# B&R Automation Studio project A2019059_Linka_Power_CP (part 26)

#### Main.st - Init, cyclic, exit code
```iecst
PROGRAM _INIT
	TprazdnyZasobnik.PT:=T#2000ms;
	TakumulaciaPlna.PT:=T#1000ms;
	TvytvorenieVakua.PT:=T#200ms;
	TodvetranieVakua.PT:=T#200ms;
	ToneskorenieVysunutia.PT:= T#500ms;
	ToneskorenieZasunutia.PT:= T#500ms;
	TvyfukovaniePredVibrovanim.PT:= T#1000ms;
    Tvibrovanie.PT:=T#3000ms;
    Stav_MaticaPripravena:= FALSE;
    TpodaniaSkrutky.PT:= T#1000ms;
    TpredMaticaPripravena.PT:= T#1000ms;
    TpripravaMatice.PT:= T#2000ms;
    TvypnutieOfuku.PT:= T#2000ms;
END_PROGRAM

PROGRAM _CYCLIC
	(********************Mapovanie IN/OUT********************************)

	SkrutkovaciSet.Manual:= P2_SkrutkovacMatic.SkrutkovaciSet_MaticaM4.Manual;
	SkrutkovaciSet.Automat:= P2_SkrutkovacMatic.SkrutkovaciSet_MaticaM4.Automat;
	SkrutkovaciSet.SkrutkaOdobrata:= P2_SkrutkovacMatic.SkrutkovaciSet_MaticaM4.MaticaM4_Odobrata;
	P2_SkrutkovacMatic.SkrutkovaciSet_MaticaM4.MaticaM4_Pripravena:= SkrutkovaciSet.SkrutkaPripravena;

	SkrutkovaciSet.Vreteno.IN.DeptControl;
	SkrutkovaciSet.Vreteno.IN.PushClinderAR:= P2_SkrutkovacMatic.IN.DavkMatic_VYSUNUTY_IS26;
	SkrutkovaciSet.Vreteno.IN.PushClinderGR:= P2_SkrutkovacMatic.IN.DavkMatic_ZASUNUTY_IS25;
	SkrutkovaciSet.Vreteno.IN.ReturnStroke:= P2_SkrutkovacMatic.IN.SkrutkMatic_ZASUNUTY_MS9;
	SkrutkovaciSet.Vreteno.IN.ScrewControl:= P2_SkrutkovacMatic.IN.DavkMatic_PritomnostMatice_OS2;
	SkrutkovaciSet.Vreteno.IN.ScrewMeasurement:= P2_SkrutkovacMatic.IN.OddelMatic_MaticaPresla_IS24;
	SkrutkovaciSet.Vreteno.IN.ScrewMeasurementPushCylinder:= P2_SkrutkovacMatic.IN.DavkMatic_MaticaPresla_IS27;

	P2_SkrutkovacMatic.OUT.PosuvacMatic_PosunMaticu_YV68:=SkrutkovaciSet.Vreteno.OUT.PushCylinder;

	SkrutkovaciSet.Zasobnik.IN.AccumulationSwitch:= P2_SkrutkovacMatic.IN.ZasobMatic_ListaPLNA_OS1;
	SkrutkovaciSet.Zasobnik.IN.FeederLevelControl:= P2_SkrutkovacMatic.IN.ZasobMatic_PRAZDNY_IS23;
	SkrutkovaciSet.Zasobnik.IN.EscapementAR:= P2_SkrutkovacMatic.IN.OddelMatic_Otoceny_VPRED_MS59;
	SkrutkovaciSet.Zasobnik.IN.EscapementGR:= P2_SkrutkovacMatic.IN.OddelMatic_Otoceny_VZAD_MS58;

	P2_SkrutkovacMatic.OUT.ZasobMatic_Ofuk_RUN_YV63:=SkrutkovaciSet.Zasobnik.OUT.BlowOff;
	P2_SkrutkovacMatic.OUT.OddelMatic_PosunMaticu_YV69:=SkrutkovaciSet.Zasobnik.OUT.Escapement;
	P2_SkrutkovacMatic.OUT.OddelMatic_NastrelMaticu_YV65:=SkrutkovaciSet.Zasobnik.OUT.FeedAir;
	P2_SkrutkovacMatic.OUT.ZasobMatic_OfukTried_RUN_YV64:=SkrutkovaciSet.Zasobnik.OUT.SortingAir;
	P2_SkrutkovacMatic.OUT.ZasobMatic_Vibrovanie_RUN_FM1:=SkrutkovaciSet.Zasobnik.OUT.StartA20;

	IF P2_SkrutkovacMatic.SkrutkovaciSet_MaticaM4.Reset THEN
		SkrutkovaciSet.VretenoFaza:=0;
		P2_SkrutkovacMatic.SkrutkovaciSet_MaticaM4.Reset:= FALSE;
	END_IF

	(********************Časáky********************************)
	TprazdnyZasobnik();
	TakumulaciaPlna();
	TvytvorenieVakua();
	TodvetranieVakua();
	ToneskorenieVysunutia();
    ToneskorenieZasunutia();
    Tvibrovanie();
    TvyfukovaniePredVibrovanim();
    TpodaniaSkrutky();
    TpredMaticaPripravena();
    TpripravaMatice();
    TvypnutieOfuku();
	(********************Zásobnik********************************)

	//kontrola akumulacie
	IF SkrutkovaciSet.Zasobnik.IN.AccumulationSwitch=1 THEN
		TakumulaciaPlna.IN:=1;
	ELSE
		TakumulaciaPlna.IN:=0;
	END_IF

	//kontrola naplnenia zasobnika
	IF SkrutkovaciSet.Zasobnik.IN.FeederLevelControl=1 THEN
		TprazdnyZasobnik.IN:=1;
	ELSE
		TprazdnyZasobnik.IN:=0;
	END_IF

    IF ZapniHrniec THEN
        TvyfukovaniePredVibrovanim.IN:= 1;
    ELSE
		TvyfukovaniePredVibrovanim.IN:= 0;
	END_IF

	IF ZapniHrniec AND TvyfukovaniePredVibrovanim.Q THEN
        SkrutkovaciSet.Zasobnik.OUT.StartA20:=1;
        Tvibrovanie.IN:=1;
	ELSE
        SkrutkovaciSet.Zasobnik.OUT.StartA20:=0;
        Tvibrovanie.IN:=0;
	END_IF

    IF Tvibrovanie.Q=1 THEN
        IF TakumulaciaPlna.Q=1 AND NOT P2_SkrutkovacMatic.RR_ZapniHrniec THEN
            ZapniHrniec:= 0;
        END_IF
    END_IF

    //Zapnutie hrnca v ručnom režime//
    IF EDGEPOS(P2_SkrutkovacMatic.RR_ZapniHrniec) THEN
        ZapniHrniec:= TRUE;
    END_IF
    IF EDGENEG(P2_SkrutkovacMatic.RR_ZapniHrniec) THEN
        ZapniHrniec:= FALSE;
    END_IF

    //Ovládanie vzduchov zásobníka//
    IF ZapniHrniec THEN
        IF TakumulaciaPlna.Q=1 THEN
            SkrutkovaciSet.Zasobnik.OUT.BlowOff:=1;
        ELSE
            SkrutkovaciSet.Zasobnik.OUT.BlowOff:=0;
        END_IF
        SkrutkovaciSet.Zasobnik.OUT.SortingAir:= 1;
    ELSE
        SkrutkovaciSet.Zasobnik.OUT.BlowOff:=0;
    END_IF

    IF NOT SkrutkovaciSet.Zasobnik.OUT.StartA20 AND NOT ZapniHrniec THEN
        TvypnutieOfuku.IN:= 1;
    ELSE
        TvypnutieOfuku.IN:= 0;
    END_IF

    IF EDGEPOS(TvypnutieOfuku.Q) THEN
        SkrutkovaciSet.Zasobnik.OUT.SortingAir:= 0;
    END_IF

	(********************Vreteno********************************)
	CASE SkrutkovaciSet.VretenoFaza OF
		0: SkrutkovaciSet.VretenoStatus:="Vypnute";
			SkrutkovaciSet.Vreteno.OUT.CounterBlast:=0;
			SkrutkovaciSet.Vreteno.OUT.Spindle:=0;

			SkrutkovaciSet.Zasobnik.OUT.Escapement:=0;
			SkrutkovaciSet.Zasobnik.OUT.FeedAir:=0;

			SkrutkovaciSet.Zasobnik.OUT.StartA20:=0;

			SkrutkovaciSet.SkrutkaPripravena:=0;

			TprazdnyZasobnik.IN:=0;
			TakumulaciaPlna.IN:=0;
			TvytvorenieVakua.IN:=0;
			TodvetranieVakua.IN:=0;
			ToneskorenieVysunutia.IN:=0;
            ToneskorenieZasunutia.IN:= 0;
            TpodaniaSkrutky.IN:= 0;
            TpredMaticaPripravena.IN:= 0;
            TpripravaMatice.IN:= 0;
			ZapniHrniec:= 0;
			SkrutkovaciSet.VretenoFaza:=1;

		1: SkrutkovaciSet.VretenoStatus:="Inicializacia: cakam na povel";
			IF SkrutkovaciSet.Automat=1 THEN
				SkrutkovaciSet.SkrutkaPripravena:=0;
				SkrutkovaciSet.VretenoFaza:=2;
			ELSIF SkrutkovaciSet.Manual=1 THEN
				SkrutkovaciSet.VretenoFaza:=250;
			ELSIF P2_SkrutkovacMatic.RR_PodajMaticu THEN
				Stav_MaticaPripravena:= FALSE;
				SkrutkovaciSet.VretenoFaza:=2;
			END_IF

		2: SkrutkovaciSet.VretenoStatus:="Inicializacia: cakam na snimac koliska vo vstupnej polohe";
			SkrutkovaciSet.Zasobnik.OUT.Escapement:=0;
			IF SkrutkovaciSet.Zasobnik.IN.EscapementGR=1 THEN
				SkrutkovaciSet.Zasobnik.OUT.FeedAir:=1;
				SkrutkovaciSet.VretenoFaza:=3;
			END_IF

		3: SkrutkovaciSet.VretenoStatus:="Inicializacia: Cakam na snimac: podavaci piest zasunuty";
			SkrutkovaciSet.Vreteno.OUT.PushCylinder:=0;
			IF SkrutkovaciSet.Vreteno.IN.PushClinderGR=1 THEN
				SkrutkovaciSet.VretenoFaza:=4;
			END_IF

		4: SkrutkovaciSet.VretenoStatus:="Inicializacia: kontrolujem pritomnost matky";
			IF SkrutkovaciSet.Vreteno.IN.ScrewControl=1 THEN
				SkrutkovaciSet.Zasobnik.OUT.FeedAir:=0;
				SkrutkovaciSet.VretenoFaza:=100;
			ELSE
				SkrutkovaciSet.VretenoFaza:=5;
			END_IF

		5: SkrutkovaciSet.VretenoStatus:="Inicializacia: Cakam na snimac: podavaci piest vysunuty";
			SkrutkovaciSet.Vreteno.OUT.PushCylinder:=1;
			IF SkrutkovaciSet.Vreteno.IN.PushClinderAR=1 THEN
				SkrutkovaciSet.VretenoFaza:=6;
			END_IF

		6: SkrutkovaciSet.VretenoStatus:="Inicializacia: Cakam na snimac: podavaci piest zasunuty";
			SkrutkovaciSet.Vreteno.OUT.PushCylinder:=0;
			IF SkrutkovaciSet.Vreteno.IN.PushClinderGR=1 THEN
				SkrutkovaciSet.VretenoFaza:=7;
			END_IF

		7: SkrutkovaciSet.VretenoStatus:="Inicializacia: kontrolujem pritomnost matky";
			IF SkrutkovaciSet.Vreteno.IN.ScrewControl=1 THEN
				SkrutkovaciSet.Vreteno.OUT.Vacuum:=1;
				SkrutkovaciSet.Zasobnik.OUT.FeedAir:=0;
				SkrutkovaciSet.VretenoFaza:=100;
			ELSE
				SkrutkovaciSet.Zasobnik.OUT.FeedAir:=0;
				SkrutkovaciSet.VretenoFaza:=150;
			END_IF

		100: SkrutkovaciSet.VretenoStatus:="Pripravene: cakam na povel";
			SkrutkovaciSet.SkrutkaPripravena:=1;
			IF P2_SkrutkovacMatic.RR_PodajMaticu THEN
				SkrutkovaciSet.Vreteno.OUT.Vacuum:=0;
				SkrutkovaciSet.SkrutkaPripravena:=0;
				P2_SkrutkovacMatic.RR_PodajMaticu:= FALSE;
                SkrutkovaciSet.VretenoFaza:=0;
			END_IF

			IF SkrutkovaciSet.SkrutkaOdobrata=1 THEN
				SkrutkovaciSet.Vreteno.OUT.Vacuum:=0;
				SkrutkovaciSet.SkrutkaPripravena:=0;
				SkrutkovaciSet.VretenoFaza:=101;
			END_IF

		101: SkrutkovaciSet.VretenoStatus:="Cakam kym zmizne signal skrutka odobrata";
			SkrutkovaciSet.SkrutkaPripravena:=0;
			IF SkrutkovaciSet.SkrutkaOdobrata=0 THEN
				SkrutkovaciSet.VretenoFaza:=150;
			END_IF

		150: SkrutkovaciSet.VretenoStatus:="Cakam kym zasobnik pripravy skrutku";
			ZapniHrniec:= 1;
            IF TakumulaciaPlna.Q=1 AND SkrutkovaciSet.Zasobnik.OUT.StartA20 THEN
                TpodaniaSkrutky.IN:= 1;
            END_IF

            IF TpodaniaSkrutky.Q THEN
                TpodaniaSkrutky.IN:= 0;
                SkrutkovaciSet.VretenoFaza:=151;
			END_IF

		151: SkrutkovaciSet.VretenoStatus:="Cakam na snimac: koliska vo vystupnej polohe";
			SkrutkovaciSet.Zasobnik.OUT.Escapement:=1;
			IF SkrutkovaciSet.Zasobnik.IN.EscapementAR=1 THEN
				SkrutkovaciSet.VretenoFaza:=152;
			END_IF

		152: SkrutkovaciSet.VretenoStatus:="Cakam na snimac: skrutka presla hadicou za zasobnikom";

            TpripravaMatice.IN:=1;
			IF SkrutkovaciSet.Vreteno.IN.ScrewMeasurement=1 THEN
                SkrutkovaciSet.Zasobnik.OUT.FeedAir:=1;
                TpripravaMatice.IN:=0;
                SkrutkovaciSet.VretenoFaza:=153;
            ELSIF TpripravaMatice.Q THEN
                TpripravaMatice.IN:=0;
                SkrutkovaciSet.Zasobnik.OUT.Escapement:=0;
                SkrutkovaciSet.VretenoFaza:=150;
			END_IF

		153: SkrutkovaciSet.VretenoStatus:="Cakam na snimac: skrutka presla hadicou pred piestom";
			SkrutkovaciSet.Zasobnik.OUT.FeedAir:=1;
			IF SkrutkovaciSet.Vreteno.IN.ScrewMeasurementPushCylinder=1 THEN
				ToneskorenieVysunutia.IN:= 1;
			END_IF
			IF ToneskorenieVysunutia.Q THEN
				ToneskorenieVysunutia.IN:= 0;
				SkrutkovaciSet.Zasobnik.OUT.FeedAir:=0;
				SkrutkovaciSet.VretenoFaza:=154;
			END_IF

		154: SkrutkovaciSet.VretenoStatus:="Cakam na snimac: podavaci piest vysunuty";
			SkrutkovaciSet.Vreteno.OUT.PushCylinder:=1;
			SkrutkovaciSet.Vreteno.OUT.Vacuum:=1;
			IF SkrutkovaciSet.Vreteno.IN.PushClinderAR=1 THEN
				SkrutkovaciSet.Zasobnik.OUT.FeedAir:=0;
				SkrutkovaciSet.VretenoFaza:=155;
			END_IF

		155: SkrutkovaciSet.VretenoStatus:="Cakam na snimac: matka v hlavici";
			ToneskorenieZasunutia.IN:= SkrutkovaciSet.Vreteno.IN.ScrewControl;
			IF SkrutkovaciSet.Vreteno.IN.ScrewControl=1 AND ToneskorenieZasunutia.Q THEN
				ToneskorenieZasunutia.IN:= 0;
				SkrutkovaciSet.VretenoFaza:=156;
			END_IF

		156: SkrutkovaciSet.VretenoStatus:="Cakam na snimac: podavaci piest zasunuty";
			SkrutkovaciSet.Vreteno.OUT.PushCylinder:=0;
			IF SkrutkovaciSet.Vreteno.IN.PushClinderGR=1 THEN
				SkrutkovaciSet.VretenoFaza:=157;
			END_IF

		157: SkrutkovaciSet.VretenoStatus:="Cakam na snimac: koliska vo vstupnej polohe";
			SkrutkovaciSet.Zasobnik.OUT.Escapement:=0;
			IF SkrutkovaciSet.Zasobnik.IN.EscapementGR=1 THEN
				SkrutkovaciSet.VretenoFaza:=158;
			END_IF

		158: SkrutkovaciSet.VretenoStatus:="Novy cyklus";
			SkrutkovaciSet.VretenoFaza:=100;
	END_CASE

END_PROGRAM

PROGRAM _EXIT
	(* Insert code here *)

END_PROGRAM
```

#### Types.typ - Local data types
```iecst
TYPE
	SkrutkovaciSetStruc : 	STRUCT
		VretenoStatus : WSTRING[80];
		VretenoFaza : USINT;
		Zasobnik : ZasobnikStruc;
		Vreteno : VretenoStruc;
		SkrutkaOdobrata : BOOL;
		SkrutkaPripravena : BOOL;
		Manual : BOOL;
		PodajSrobu : BOOL;
		CistenieVykonane : BOOL;
		VykonajCistenie : BOOL;
		Automat : BOOL;
	END_STRUCT;
	INzasobnik : 	STRUCT
		EscapementGR : BOOL;
		EscapementAR : BOOL;
		AccumulationSwitch : BOOL; (*Snimac zaplnenia S25*)
		FeederLevelControl : BOOL; (*Hladina v zasobniku S20*)
	END_STRUCT;
	OUTzasobnik : 	STRUCT
		StartA20 : BOOL; (*Zapnutie vibrovania A20*)
		Escapement : BOOL; (*Pustanie matky do hadice Y22*)
		FeedAir : BOOL; (*Strielanie do hadice Y21*)
		SortingAir : BOOL; (*Triedenie kusov Y30*)
		BlowOff : BOOL; (*Zhadzovanie kusov Y25*)
	END_STRUCT;
	INvreteno : 	STRUCT
		ReturnStroke : BOOL; (*Vreteno zasunute S01*)
		DeptControl : BOOL; (*Vreteno vysunute S02*)
		PushClinderGR : BOOL; (*Posuvaci valec v domovskej  polohe S11*)
		PushClinderAR : BOOL; (*Posuvaci valec v pracovnej polohe S10*)
		ScrewMeasurement : BOOL; (*Kontrola matice v hadici S21*)
		ScrewMeasurementPushCylinder : BOOL; (*Kontrola matice v posuvacom valci S06*)
		ScrewControl : BOOL; (*Kontrola matice vo vretene S14*)
	END_STRUCT;
	OUTvreteno : 	STRUCT
		Spindle : BOOL; (*Vysunutie vretena Y02*)
		Vacuum : BOOL; (*Pridrzanie skrutky Y15*)
		PushCylinder : BOOL; (*Posunutie z hadice do hlavy Y10*)
		CounterBlast : BOOL; (*Uvolnenie skrutky Y16*)
	END_STRUCT;
	VretenoStruc : 	STRUCT
		OUT : OUTvreteno;
		IN : INvreteno;
	END_STRUCT;
	ZasobnikStruc : 	STRUCT
		OUT : OUTzasobnik;
		IN : INzasobnik;
	END_STRUCT;
END_TYPE
```

#### Variables.var - Local variables
```iecst
VAR
	TvytvorenieVakua : TON;
	TodvetranieVakua : TON;
	TprazdnyZasobnik : TON;
	TakumulaciaPlna : TON;
	ToneskorenieVysunutia : TON;
	ToneskorenieZasunutia : TON;
	SkrutkovaciSet : SkrutkovaciSetStruc;
	Stav_MaticaPripravena : BOOL;
	TvyfukovaniePredVibrovanim : TON;
	ZapniHrniec : BOOL;
	TpodaniaSkrutky : TON;
	Tvibrovanie : TON;
	TpredMaticaPripravena : TON;
	TpripravaMatice : TON;
	TvypnutieOfuku : TON;
END_VAR
```

### Program Logical/Program/Pracovisko_2/P2_StoperSrobovania (IEC)

#### Main.st - Init, cyclic, exit code
```iecst
PROGRAM _INIT
    Triger_0:= FALSE;
    Triger_1:= FALSE;

END_PROGRAM

PROGRAM _CYCLIC

	//Volanie funkcie SequenceControl//
    SequenceControl(SC:= SC_P2_StoperSrobovania);

    //Volanie podprogramov//
    OvlCentrovacky;
    IOLinkKomunikacia;

    //Reset sekcie //
    IF P2_StoperSrobovania.Reset THEN
        SC_P2_StoperSrobovania.Step:= 0;
        P2_StoperSrobovania.Reset:= FALSE;
    END_IF

    IF NOT Safety.STAV.P2_ZonaBunky_AKTIVNA AND NOT P2_StoperSrobovania.Automat THEN
        SC_P2_StoperSrobovania.Step:= 0;
    END_IF

    IF NOT Safety.STAV.P2_ZonaBunky_AKTIVNA AND NOT Triger_0 THEN
        Triger_0:= TRUE;
        IF P2_StoperSrobovania.IN.PritomnostPaletky_S8 AND P2_StoperSrobovania.Automat THEN
            IF NOT Paletka[i].VnutornyStav.KomunikaciaOtvorena THEN
                SC_P2_StoperSrobovania.ResetStep:= TRUE;
                SC_P2_StoperSrobovania.Step:= 0;
            ELSIF Paletka[i].VnutornyStav.KomunikaciaUzavreta THEN
                SC_P2_StoperSrobovania.ResetStep:= TRUE;
                SC_P2_StoperSrobovania.Step:= 0;
            ELSIF Paletka[i].VnutornyStav.CinnostSpustena THEN
                Paletka[i].PAR.StavPowerCP:= 'FAIL';
                Paletka[i].PAR.StavPaletky:= 'NG';
                P2_StoperSrobovania.KoniecCyklu:= TRUE;
                SC_P2_StoperSrobovania.ResetStep:= TRUE;
                SC_P2_StoperSrobovania.Step:= 550;
            ELSIF Paletka[i].VnutornyStav.KomunikaciaOtvorena THEN
                Paletka[i].PAR.StavPowerCP:= 'FAIL';
                Paletka[i].PAR.StavPaletky:= 'NG';
                P2_StoperSrobovania.KoniecCyklu:= TRUE;
                SC_P2_StoperSrobovania.ResetStep:= TRUE;
                SC_P2_StoperSrobovania.Step:= 550;
            END_IF
        END_IF
    END_IF

    IF Safety.STAV.P2_ZonaBunky_AKTIVNA THEN
        Triger_0:= FALSE;
    END_IF

    //Porucha stanice//
    IF P2_PoruchaST3 AND NOT Triger_1 THEN
        Triger_1:= TRUE;
        IF P2_StoperSrobovania.IN.PritomnostPaletky_S8 AND P2_StoperSrobovania.Automat THEN
            SC_P2_Srobovanie.Step:= 0;
            IF NOT Paletka[i].VnutornyStav.KomunikaciaOtvorena THEN
                SC_P2_StoperSrobovania.ResetStep:= TRUE;
                SC_P2_StoperSrobovania.Step:= 0;
            ELSIF Paletka[i].VnutornyStav.KomunikaciaUzavreta THEN
                SC_P2_StoperSrobovania.ResetStep:= TRUE;
                SC_P2_StoperSrobovania.Step:= 0;
            ELSIF Paletka[i].VnutornyStav.CinnostSpustena THEN
                Paletka[i].PAR.StavPowerCP:= 'FAIL';
                Paletka[i].PAR.StavPaletky:= 'NG';
                P2_StoperSrobovania.KoniecCyklu:= TRUE;
                SC_P2_StoperSrobovania.ResetStep:= TRUE;
                SC_P2_StoperSrobovania.Step:= 550;
            ELSIF Paletka[i].VnutornyStav.KomunikaciaOtvorena THEN
                Paletka[i].PAR.StavPowerCP:= 'FAIL';
                Paletka[i].PAR.StavPaletky:= 'NG';
                P2_StoperSrobovania.KoniecCyklu:= TRUE;
                SC_P2_StoperSrobovania.ResetStep:= TRUE;
                SC_P2_StoperSrobovania.Step:= 550;
            END_IF
        ELSE
            SC_P2_StoperSrobovania.ResetStep:= TRUE;
            SC_P2_StoperSrobovania.Step:= 0;
        END_IF
    END_IF

    IF NOT P2_PoruchaST3 THEN
        Triger_1:= FALSE;
    END_IF

    CASE SC_P2_StoperSrobovania.Step OF

        0:
            SC_P2_StoperSrobovania.StepName:='0 - Nulovanie';
            SC_OvlCentrovacky.Step:= 0;
            P2_StoperSrobovania.Automat:= FALSE;
            P2_StoperSrobovania.KoniecCyklu:= FALSE;
            P2_StoperSrobovania.Manual:= FALSE;
            P2_StoperSrobovania.STAV.PoINIT:= FALSE;
            P2_StoperSrobovania.OUT.ZasunStoper_YV56:= FALSE;
            P2_StoperSrobovania.OUT.KOM_4F_ZasrobujLavuSkrutkuM4:= FALSE;
            P2_StoperSrobovania.OUT.KOM_4F_ZasrobujPravuSkrutkuM4:= FALSE;
            P2_StoperSrobovania.OUT.KOM_4F_ZasrobujLavuSkrutkuM6:= FALSE;
            P2_StoperSrobovania.OUT.KOM_4F_ZasrobujPravuSkrutkuM6:= FALSE;
            P2_StoperSrobovania.OUT.KOM_5F_ZasrobujLavuSkrutkuM4:= FALSE;
            P2_StoperSrobovania.OUT.KOM_5F_ZasrobujPravuSkrutkuM4:= FALSE;
            P2_StoperSrobovania.OUT.KOM_5F_ZasrobujLavuSkrutkuM6:= FALSE;
            P2_StoperSrobovania.OUT.KOM_5F_ZasrobujPravuSkrutkuM6:= FALSE;
            P2_StoperSrobovania.OUT.KOM_5H_ZasrobujLavuSkrutkuM5:= FALSE;
            P2_StoperSrobovania.OUT.KOM_5H_ZasrobujPravuSkrutkuM5:= FALSE;
            P2_StoperSrobovania.OUT.KOM_5H_ZasrobujSkrutkuM4:= FALSE;
            P2_StoperSrobovania.OUT.KOM_PresunManipulator_DOPREDU:= FALSE;
            P2_StoperSrobovania.OUT.KOM_PresunManipulator_DOZADU:= FALSE;
            P2_Srobovanie.OUT.KOM_Srobovanie_Ukoncene:= FALSE;
            P2_Srobovanie.OUT.KOM_PresunVPRED_Ukonceny:= FALSE;
            P2_Srobovanie.OUT.KOM_PresunVZAD_Ukonceny:= FALSE;
            P2_Robot.KOM_OUT.Odober_Busbary4F:= FALSE;
            P2_Robot.KOM_OUT.Odober_Busbary5F:= FALSE;
            P2_Robot.KOM_OUT.Odober_Busbary5H:= FALSE;
            P2_Robot.KOM_OUT.Poloz_Busbary4F:= FALSE;
            P2_Robot.KOM_OUT.Poloz_Busbary5F:= FALSE;
            P2_Robot.KOM_OUT.Poloz_Busbary5H:= FALSE;
            P2_Robot.KOM_OUT.Dotlac_Filter5H:= FALSE;
            P2_Robot.KOM_OUT.Odparkovanie:= FALSE;
            P2_Robot.KOM_OUT.Presun_CakaciaPozicia:= FALSE;
            P2_Robot.KOM_OUT.UvolniBusbary:= FALSE;
            P2_Robot.KOM_OUT.Dotlac_Filter5H:= FALSE;
            P2_Robot.KOM_OUT.ZmenaGripra_Cistenie:= FALSE;
            CAM10.CMD.Triger:= FALSE;
            CAM10.STAV.Results_READY:= FALSE;
            FTP_CAM10.CMD.OdosliFotku:= FALSE;
            FTP_CAM10.CMD.VymazFotku:= FALSE;
            P2_StoperSrobovania.STAV.KOM_PLC_OdoslanieFotiek_OK:= FALSE;
            P2_StoperSrobovania.STAV.KOM_PLC_VymazanieFotiek_OK:= FALSE;
            TRCB_P2_Srobovanie_ST5.CMD.VyziadajStavPaletky_TYP1:= FALSE;
            TRCB_P2_Srobovanie_ST5.CMD.PriradQRkodFiltra_TYP3:= FALSE;
            TRCB_P2_Srobovanie_ST5.CMD.OdosliStavPaletky_TYP2:= FALSE;
            PrecitaneCisloPaletky:= '';
            P2_Srobov_ManipulaciaUkoncena:= FALSE;
            PocetDopytovNaServer:= 0;
            Taktime_Srobovanie_ST5.CMD.START_Merania_1:= FALSE;
            Taktime_Srobovanie_ST5.CMD.START_Merania_2:= FALSE;
            P2_StoperSrobovania.STAV.PrebiehaVyvezeniePaletky:= FALSE;
            P2_Srobov_KAM_Result_Ignoruj:= FALSE;
            P2_Srobov_CakaNaKameru:= FALSE;
            P2_StoperSrobovania.STAV.Porucha:= FALSE;
            TestovaciKus:= FALSE;
            Revork:= FALSE;
            P2_Robot.STAV.Srobovanie_PrebiehaManipulacia:= FALSE;
            CisloFotky:= 0;
            P2_Srobov_KAM_Result_OK:= FALSE;
            P2_Srobov_KAM_Result_NG:= FALSE;
            P2_Vizu.ZobrazHL1_ST5:= FALSE;
            P2_Vizu.ZobrazHL2_ST5:= FALSE;
            P2_Vizu.ZobrazHL3_ST5:= FALSE;
            P2_Vizu.ZobrazHL4_ST5:= FALSE;
            TRCB_P2_Srobov_OpatovnyDopyt:= FALSE;
            TRCB_P2_Srobov_PaletkaNG:= FALSE;
            VysunutieSkrutkovacky_OK:= FALSE;
            PocetTrigrovKamery:= 0;
            DoskrutkovaniePriPoruche:= FALSE;

            IF Safety.STAV.P2_ZonaBunky_AKTIVNA AND NOT P2_Pracovisko.STAV.PORUCHA AND P2_Pracovisko.IN.PrivodVzduchu_SnimacTlaku_S3 THEN
                SC_P2_StoperSrobovania.ResetStep:= TRUE;
                SC_P2_StoperSrobovania.Step:= 1;
            END_IF

        1:
            SC_P2_StoperSrobovania.StepName:='1 - Cakam na spustenie vyroby';
            P2_StoperSrobovania.KoniecCyklu:= FALSE;
            IF P2_StoperSrobovania.Automat THEN
                SC_P2_StoperSrobovania.Step:= 2;
            ELSIF P2_StoperSrobovania.Manual THEN
                SC_P2_StoperSrobovania.Step:= 700;
            END_IF

            //********************************************************Inicializácia****************************************************************************//

        2:
            SC_P2_StoperSrobovania.StepName:='2 - Inicializacia - cakam na spustenie inicializacie';
            SC_P2_StoperSrobovania.IdleTime.PT:= T#4s;
            SC_P2_StoperSrobovania.AlarmTime.PT:= T#5s;

            IF P2_Srobovanie.STAV.PoINIT AND P2_Srobovacky_VychodziaPozicia THEN
                SC_P2_StoperSrobovania.ResetStep:= TRUE;
                SC_P2_StoperSrobovania.Step:= 3;
            END_IF

        3:
            SC_P2_StoperSrobovania.StepName:='3 - Inicializacia - vymazanie adresara kamery';
            SC_P2_StoperSrobovania.IdleTime.PT:= T#4s;
            SC_P2_StoperSrobovania.AlarmTime.PT:= T#5s;

            IF NOT SC_P2_StoperSrobovania.Switch1 THEN
                FTP_CAM10.CMD.VymazFotku:= TRUE;
                SC_P2_StoperSrobovania.Switch1:= TRUE;
            END_IF

            IF FTP_CAM10.STATUS.KomunikaciaUkoncena THEN
                FTP_CAM10.CMD.VymazFotku:= FALSE;
                SC_P2_StoperSrobovania.ResetStep:= TRUE;
                SC_P2_StoperSrobovania.Step:= 5;
            ELSIF FTP_CAM10.STATUS.KomunikaciaError THEN
                P2_Alarmy[232]:= TRUE;
                P2_PoruchaST3:= TRUE;
            END_IF

        5:
            SC_P2_StoperSrobovania.StepName:='5 - Inicializacia - kontrola pozicie robota';
            SC_P2_StoperSrobovania.IdleTime.PT:= T#5s;
            SC_P2_StoperSrobovania.AlarmTime.PT:= T#5s;

            IF P2_Robot.KOM_IN.Stav_RobotBezpPozicia_Srobovanie THEN
                SC_P2_StoperSrobovania.ResetStep:= TRUE;
                SC_P2_StoperSrobovania.Step:= 10;
            END_IF

        10:
            SC_P2_StoperSrobovania.StepName:='10 - Inicializacia - zasunutie centrovacky';
            SC_P2_StoperSrobovania.IdleTime.PT:= T#4s;
            SC_P2_StoperSrobovania.AlarmTime.PT:= T#5s;

            IF NOT SC_P2_StoperSrobovania.Switch1 THEN
                Centrovacku_ZASUN:= TRUE;
                SC_P2_StoperSrobovania.Switch1:= TRUE;
            END_IF

            IF P2_StoperSrobovania.IN.Centrovanie_ZASUNUTE_IS15 AND P2_Dopravniky.STAV.PoINIT THEN
                SC_P2_StoperSrobovania.ResetStep:= TRUE;
                SC_P2_StoperSrobovania.Step:= 13;
            END_IF

        13:
            SC_P2_StoperSrobovania.StepName:='13 - Inicializacia - hladanie paletky';
            SC_P2_StoperSrobovania.IdleTime.PT:= T#5s;
            SC_P2_StoperSrobovania.AlarmTime.PT:= T#5s;
            SC_P2_StoperSrobovania.IdleTime.IN:= TRUE;

            IF P2_StoperSrobovania.IN.PritomnostPaletky_S8 THEN
                P2_StoperMaticovacky.STAV.PrebiehaVyvezeniePaletky:= FALSE;
                SC_P2_StoperSrobovania.ResetStep:= TRUE;
                SC_P2_StoperSrobovania.Step:= 20;
            ELSIF SC_P2_StoperSrobovania.IdleTime.Q THEN
                P2_StoperSrobovania.STAV.PoINIT:= TRUE;
                SC_P2_StoperSrobovania.ResetStep:= TRUE;
                SC_P2_StoperSrobovania.Step:= 100;
            END_IF

        20:
            SC_P2_StoperSrobovania.StepName:='20 - Inicializacia - precitanie cisla paletky';
            SC_P2_StoperSrobovania.IdleTime.PT:= T#200ms;
            SC_P2_StoperSrobovania.AlarmTime.PT:= T#5s;
            SC_P2_StoperSrobovania.IdleTime.IN:= TRUE;

            IF SC_P2_StoperSrobovania.IdleTime.Q THEN
                PrecitaneCisloPaletky:= USINT_TO_STRING(P2_StoperSrobovania.IN.PrecitaneCisloPaletky_S8);
                i:= 0;
                SC_P2_StoperSrobovania.ResetStep:= TRUE;
                SC_P2_StoperSrobovania.Step:= 23;
            END_IF

        23:
            SC_P2_StoperSrobovania.StepName:='23 - Inicializacia - priradenie indexu paletky na zaklade precitanej hodnoty';
            SC_P2_StoperSrobovania.IdleTime.PT:= T#200ms;
            SC_P2_StoperSrobovania.AlarmTime.PT:= T#5s;

            IF PrecitaneCisloPaletky = '171' THEN
                i:= 1;
            ELSIF PrecitaneCisloPaletky = '164' THEN
                i:= 2;
            ELSIF PrecitaneCisloPaletky = '181' THEN
                i:= 3;
            ELSIF PrecitaneCisloPaletky = '168' THEN
                i:= 4;
            ELSIF PrecitaneCisloPaletky = '140' THEN
                i:= 5;
            ELSIF PrecitaneCisloPaletky = '110' THEN
                i:= 6;
            ELSIF PrecitaneCisloPaletky = '156' THEN
                i:= 7;
            ELSIF PrecitaneCisloPaletky = '127' THEN
                i:= 8;
            ELSIF PrecitaneCisloPaletky = '139' THEN
                i:= 9;
            ELSIF PrecitaneCisloPaletky = '131' THEN
                i:= 10;
            ELSIF PrecitaneCisloPaletky = '178' THEN
                i:= 11;
            ELSIF PrecitaneCisloPaletky = '206' THEN
                i:= 12;
            ELSIF PrecitaneCisloPaletky = '119' THEN
                i:= 13;
            ELSIF PrecitaneCisloPaletky = '163' THEN
                i:= 14;
            ELSIF PrecitaneCisloPaletky = '128' THEN
                i:= 15;
            ELSIF PrecitaneCisloPaletky = '175' THEN
                i:= 16;
            ELSIF PrecitaneCisloPaletky = '138' THEN
                i:= 17;
            ELSE
                P2_Alarmy[214]:= TRUE;
                P2_PoruchaST3:= TRUE;
            END_IF

            IF i<> 0 THEN
                Paletka[i].PAR.CisloPaletky:= USINT_TO_STRING(i);
                P2_StoperSrobovania.PAR.IndexPaletky_STRING:= USINT_TO_STRING(i);
                P2_StoperSrobovania.PAR.IndexPaletky:= i;
                PrecitaneCisloPaletky:= '';
                SC_P2_StoperSrobovania.ResetStep:= TRUE;
                SC_P2_StoperSrobovania.Step:= 30;
            END_IF

        30:
            SC_P2_StoperSrobovania.StepName:='30 - Inicializacia - kontrola stavu paletky';
            SC_P2_StoperSrobovania.IdleTime.PT:= T#200ms;
            SC_P2_StoperSrobovania.AlarmTime.PT:= T#5s;

            IF Paletka[i].PAR.TestovaciKus AND Paletka[i].PAR.CisloTestovacejStanice = 'ST_5' THEN
                TestovaciKus:= TRUE;
            ELSIF Paletka[i].PAR.TestovaciKus AND Paletka[i].PAR.CisloTestovacejStanice <> 'ST_5' THEN
                P2_StoperSrobovania.STAV.PoINIT:= TRUE;
                SC_P2_StoperSrobovania.ResetStep:= TRUE;
                SC_P2_StoperSrobovania.Step:= 560;
            ELSIF Paletka[i].PAR.RevorkovyKus AND Paletka[i].PAR.CisloRevorkovejStanice = 'ST_5' THEN
                Revork:= TRUE;
                SC_P2_StoperSrobovania.ResetStep:= TRUE;
                SC_P2_StoperSrobovania.Step:= 33;
            ELSIF Paletka[i].PAR.RevorkovyKus AND Paletka[i].PAR.CisloRevorkovejStanice <> 'ST_5' THEN
                Revork:= FALSE;
                P2_StoperSrobovania.STAV.PoINIT:= TRUE;
                SC_P2_StoperSrobovania.ResetStep:= TRUE;
                SC_P2_StoperSrobovania.Step:= 560;
            ELSIF Paletka[i].PAR.StavPaletky = 'OK' THEN
                SC_P2_StoperSrobovania.ResetStep:= TRUE;
                SC_P2_StoperSrobovania.Step:= 33;
            ELSIF Paletka[i].PAR.StavPaletky = 'NG' THEN
                P2_StoperSrobovania.STAV.PoINIT:= TRUE;
                SC_P2_StoperSrobovania.ResetStep:= TRUE;
                SC_P2_StoperSrobovania.Step:= 560;
            END_IF

        33:
            SC_P2_StoperSrobovania.StepName:='33 - Inicializacia - kontrola uzavretia komunikacie';
            SC_P2_StoperSrobovania.IdleTime.PT:= T#200ms;
            SC_P2_StoperSrobovania.AlarmTime.PT:= T#5s;

            IF Paletka[i].VnutornyStav.KomunikaciaUzavreta THEN
                P2_StoperSrobovania.STAV.PoINIT:= TRUE;
                SC_P2_StoperSrobovania.ResetStep:= TRUE;
                SC_P2_StoperSrobovania.Step:= 560;
            ELSE
                SC_P2_StoperSrobovania.ResetStep:= TRUE;
                SC_P2_StoperSrobovania.Step:= 35;
            END_IF

        35:
            SC_P2_StoperSrobovania.StepName:='35 - Inicializacia - kontrola otvorenia komunikacie';
            SC_P2_StoperSrobovania.IdleTime.PT:= T#200ms;
            SC_P2_StoperSrobovania.AlarmTime.PT:= T#5s;

            IF Paletka[i].VnutornyStav.KomunikaciaOtvorena THEN
                SC_P2_StoperSrobovania.ResetStep:= TRUE;
                SC_P2_StoperSrobovania.Step:= 38;
            ELSE
                P2_StoperSrobovania.STAV.PoINIT:= TRUE;
                SC_P2_StoperSrobovania.ResetStep:= TRUE;
                SC_P2_StoperSrobovania.Step:= 100;
            END_IF

        38:
            SC_P2_StoperSrobovania.StepName:='38 - Inicializacia - kontrola odoslania fotiek';
            SC_P2_StoperSrobovania.IdleTime.PT:= T#5s;
            SC_P2_StoperSrobovania.AlarmTime.PT:= T#5s;

            IF Paletka[i].VnutornyStav.FotkyOdoslane THEN
                P2_StoperSrobovania.STAV.PoINIT:= TRUE;
                SC_P2_StoperSrobovania.ResetStep:= TRUE;
                SC_P2_StoperSrobovania.Step:= 550;
            ELSE
                SC_P2_StoperSrobovania.ResetStep:= TRUE;
                SC_P2_StoperSrobovania.Step:= 40;
            END_IF

        40:
            SC_P2_StoperSrobovania.StepName:='40 - Inicializacia - zacentrovanie paletky';
            SC_P2_StoperSrobovania.IdleTime.PT:= T#200ms;
            SC_P2_StoperSrobovania.AlarmTime.PT:= T#5s;

            IF NOT SC_P2_StoperSrobovania.Switch1 THEN
                Centrovacku_VYSUN:= TRUE;
                SC_P2_StoperSrobovania.Switch1:= TRUE;
            END_IF

            IF P2_StoperSrobovania.IN.Centrovanie_VYSUNUTE_IS14 THEN
                SC_P2_StoperSrobovania.ResetStep:= TRUE;
                SC_P2_StoperSrobovania.Step:= 43;
            END_IF

        43:
            SC_P2_StoperSrobovania.StepName:='43 - Inicializacia - presun manipulatora vzad';
            SC_P2_StoperSrobovania.IdleTime.PT:= T#200ms;
            SC_P2_StoperSrobovania.AlarmTime.PT:= T#5s;

            IF NOT SC_P2_StoperSrobovania.Switch1 AND P2_Robot.KOM_IN.Stav_RobotBezpPozicia_Srobovanie THEN
                P2_StoperSrobovania.OUT.KOM_PresunManipulator_DOZADU:= TRUE;
                SC_P2_StoperSrobovania.Switch1:= TRUE;
            END_IF

            IF P2_Srobovanie.OUT.KOM_PresunVZAD_Ukonceny THEN
                P2_Srobovanie.OUT.KOM_PresunVZAD_Ukonceny:= FALSE;
                P2_StoperSrobovania.OUT.KOM_PresunManipulator_DOZADU:= FALSE;
                CAM10.STAV.Results_READY:= FALSE;
                SC_P2_StoperSrobovania.ResetStep:= TRUE;
                SC_P2_StoperSrobovania.Step:= 45;
            END_IF

        45:
            SC_P2_StoperSrobovania.StepName:='45 - Inicializacia - kamerova kontrola paletky'; //CAM 10//
            SC_P2_StoperSrobovania.IdleTime.PT:= T#5s;
            SC_P2_StoperSrobovania.AlarmTime.PT:= T#5s;

            IF NOT SC_P2_StoperSrobovania.Switch1 AND CAM10.STAV.Command_READY THEN
                CAM10.CMD.Triger:= TRUE;
                SC_P2_StoperSrobovania.IdleTime.IN:= TRUE;
                SC_P2_StoperSrobovania.Switch1:= TRUE;
            END_IF

            IF CAM10.STAV.Results_READY AND CAM10.STAV.Command_AKCEPTOVANY THEN
                PocetTrigrovKamery:= 0;
                CAM10.STAV.Results_READY:= FALSE;
                SC_P2_StoperSrobovania.ResetStep:= TRUE;
                SC_P2_StoperSrobovania.Step:= 50;
            ELSIF SC_P2_StoperSrobovania.IdleTime.Q AND PocetTrigrovKamery < 5 THEN
                PocetTrigrovKamery:= PocetTrigrovKamery + 1;
                CAM10.STAV.Results_READY:= FALSE;
                CAM10.CMD.Triger:= FALSE;
                SC_P2_StoperSrobovania.ResetStep:= TRUE;
                SC_P2_StoperSrobovania.Step:= 48;
            ELSIF SC_P2_StoperSrobovania.IdleTime.Q AND PocetTrigrovKamery >= 5 THEN
                P2_Alarmy[295]:= TRUE;
                P2_PoruchaST3:= TRUE;
            END_IF

        48:
            SC_P2_StoperSrobovania.StepName:='48 - Inicializacia - cakam na opatovny triger kamery';//CAM 10//
            SC_P2_StoperSrobovania.IdleTime.PT:= T#1s;
            SC_P2_StoperSrobovania.AlarmTime.PT:= T#5s;

            SC_P2_StoperSrobovania.IdleTime.IN:= TRUE;

            IF SC_P2_StoperSrobovania.IdleTime.Q THEN
                SC_P2_StoperSrobovania.ResetStep:= TRUE;
                SC_P2_StoperSrobovania.Step:= 45;
            END_IF

        50:
            SC_P2_StoperSrobovania.StepName:='50 - Inicializacia - kontrola vysledku kamery podla typu modelu';
            SC_P2_StoperSrobovania.IdleTime.PT:= T#200ms;
            SC_P2_StoperSrobovania.AlarmTime.PT:= T#5s;

            IF NOT CAM10.STAV.BUSY THEN
                CAM10.CMD.Triger:= FALSE;
                IF Linka.PAR.ZvolenyModel = '4F' THEN
                    IF CAM10.RESULT.Paletka.Pritomn_Busbarov_4F AND
                        NOT CAM10.RESULT.PowerCP.Pritomn_LavejM4_4F5F AND
                        NOT CAM10.RESULT.PowerCP.Pritomn_LavejSkrutkyM6_4F5F AND
                        NOT CAM10.RESULT.PowerCP.Pritomn_PravejM4_4F5F AND
                        NOT CAM10.RESULT.PowerCP.Pritomn_PravejSkrutkyM6_4F5F THEN
                        CAM10.PAR.ResultFotky:= 'PASS';
                        SC_P2_StoperSrobovania.ResetStep:= TRUE;
                        SC_P2_StoperSrobovania.Step:= 53;
                    ELSE
                        CAM10.PAR.ResultFotky:= 'FAIL';
                        SC_P2_StoperSrobovania.ResetStep:= TRUE;
                        SC_P2_StoperSrobovania.Step:= 53;
                    END_IF
                ELSIF Linka.PAR.ZvolenyModel = '5F' THEN
                    IF CAM10.RESULT.Paletka.Pritomn_Busbarov_5F AND
                        NOT CAM10.RESULT.PowerCP.Pritomn_LavejM4_4F5F AND
                        NOT CAM10.RESULT.PowerCP.Pritomn_LavejSkrutkyM6_4F5F AND
                        NOT CAM10.RESULT.PowerCP.Pritomn_PravejM4_4F5F AND
                        NOT CAM10.RESULT.PowerCP.Pritomn_PravejSkrutkyM6_4F5F THEN
                        CAM10.PAR.ResultFotky:= 'PASS';
                        SC_P2_StoperSrobovania.ResetStep:= TRUE;
                        SC_P2_StoperSrobovania.Step:= 53;
                    ELSE
                        CAM10.PAR.ResultFotky:= 'FAIL';
                        SC_P2_StoperSrobovania.ResetStep:= TRUE;
                        SC_P2_StoperSrobovania.Step:= 53;
                    END_IF
                ELSIF Linka.PAR.ZvolenyModel = '5H' THEN
                    IF CAM10.RESULT.Paletka.Pritomn_Busbarov_5H AND
                        NOT CAM10.RESULT.PowerCP.Pritomn_LavejSkrutkyM5_5H AND
                        NOT CAM10.RESULT.PowerCP.Pritomn_PravejSkrutkyM5_5H AND
                        NOT CAM10.RESULT.PowerCP.Pritomn_SkrutkyM4_Filtra_5H THEN
                        CAM10.PAR.ResultFotky:= 'PASS';
                        SC_P2_StoperSrobovania.ResetStep:= TRUE;
                        SC_P2_StoperSrobovania.Step:= 53;
                    ELSE
                        CAM10.PAR.ResultFotky:= 'FAIL';
                        SC_P2_StoperSrobovania.ResetStep:= TRUE;
                        SC_P2_StoperSrobovania.Step:= 53;
                    END_IF
                END_IF
            END_IF

        53:
            SC_P2_StoperSrobovania.StepName:='53 - Inicializacia - vymazanie adresara kamery';
            SC_P2_StoperSrobovania.IdleTime.PT:= T#4s;
            SC_P2_StoperSrobovania.AlarmTime.PT:= T#5s;

            IF NOT SC_P2_StoperSrobovania.Switch1 THEN
                FTP_CAM10.CMD.VymazFotku:= TRUE;
                SC_P2_StoperSrobovania.Switch1:= TRUE;
            END_IF

            IF FTP_CAM10.STATUS.KomunikaciaUkoncena THEN
                FTP_CAM10.CMD.VymazFotku:= FALSE;
                SC_P2_StoperSrobovania.ResetStep:= TRUE;
                SC_P2_StoperSrobovania.Step:= 55;
            ELSIF FTP_CAM10.STATUS.KomunikaciaError THEN
                P2_Alarmy[232]:= TRUE;
                P2_PoruchaST3:= TRUE;
            END_IF

        55:
            SC_P2_StoperSrobovania.StepName:='55 - Inicializacia - rozhodnutie podla kamerovej kontroly paletky';
            SC_P2_StoperSrobovania.IdleTime.PT:= T#200ms;
            SC_P2_StoperSrobovania.AlarmTime.PT:= T#5s;

            IF CAM10.PAR.ResultFotky = 'PASS' THEN
                P2_StoperSrobovania.STAV.PoINIT:= TRUE;
                IF Linka.PAR.ZvolenyModel = '4F' THEN
                    SC_P2_StoperSrobovania.ResetStep:= TRUE;
                    SC_P2_StoperSrobovania.Step:= 138;
                ELSIF Linka.PAR.ZvolenyModel = '5F' THEN
                    SC_P2_StoperSrobovania.ResetStep:= TRUE;
                    SC_P2_StoperSrobovania.Step:= 258;
                ELSIF Linka.PAR.ZvolenyModel = '5H' THEN
                    SC_P2_StoperSrobovania.ResetStep:= TRUE;
                    SC_P2_StoperSrobovania.Step:= 358;
                END_IF
            ELSIF CAM10.PAR.ResultFotky = 'FAIL' THEN
                P2_StoperSrobovania.STAV.PoINIT:= TRUE;
                Paletka[i].PAR.StavPowerCP:= 'FAIL';
                SC_P2_StoperSrobovania.ResetStep:= TRUE;
                SC_P2_StoperSrobovania.Step:= 545;
            END_IF

            //********************************************************Automatický režim****************************************************************************//

        100:
            SC_P2_StoperSrobovania.StepName:='100 - Automaticky Rezim - cakam na príchod paletky na stoper';
            SC_P2_StoperSrobovania.IdleTime.PT:= T#200ms;
            SC_P2_StoperSrobovania.AlarmTime.PT:= T#5s;

            IF P2_StoperSrobovania.IN.PritomnostPaletky_S8 THEN
                P2_Robot.STAV.Srobovanie_PrebiehaManipulacia:= TRUE;
                P2_StoperMaticovacky.STAV.PrebiehaVyvezeniePaletky:= FALSE;
            END_IF

            SC_P2_StoperSrobovania.IdleTime.IN:= P2_StoperSrobovania.IN.PritomnostPaletky_S8;

            IF EDGEPOS(P2_StoperSrobovania.IN.PritomnostPaletky_S8)THEN
                IF NOT Taktime_Srobovanie_ST5.CMD.START_Merania_1 THEN
                    Taktime_Srobovanie_ST5.CMD.START_Merania_1:= TRUE;
                ELSE
                    Taktime_Srobovanie_ST5.CMD.ZAPIS_Hodnot_1:= TRUE;
                END_IF
            END_IF

            IF P2_StoperSrobovania.KoniecCyklu THEN
                SC_P2_StoperSrobovania.ResetStep:= TRUE;
                SC_P2_StoperSrobovania.Step:= 0;
            ELSIF SC_P2_StoperSrobovania.IdleTime.Q THEN
                SC_P2_StoperSrobovania.ResetStep:= TRUE;
                SC_P2_StoperSrobovania.Step:= 101;
            END_IF

        101:
            SC_P2_StoperSrobovania.StepName:='101 - Automaticky Rezim - precitanie cisla paletky';
            SC_P2_StoperSrobovania.IdleTime.PT:= T#500ms;
            SC_P2_StoperSrobovania.AlarmTime.PT:= T#5s;
            SC_P2_StoperSrobovania.IdleTime.IN:= TRUE;

            PrecitaneCisloPaletky:= USINT_TO_STRING(P2_StoperSrobovania.IN.PrecitaneCisloPaletky_S8);
            i:= 0;
            SC_P2_StoperSrobovania.ResetStep:= TRUE;
            SC_P2_StoperSrobovania.Step:= 103;

        103:
            SC_P2_StoperSrobovania.StepName:='103 - Automaticky Rezim - priradenie indexu paletky na zaklade precitanej hodnoty';
            SC_P2_StoperSrobovania.IdleTime.PT:= T#200ms;
            SC_P2_StoperSrobovania.AlarmTime.PT:= T#5s;

            IF PrecitaneCisloPaletky = '171' THEN
                i:= 1;
            ELSIF PrecitaneCisloPaletky = '164' THEN
                i:= 2;
            ELSIF PrecitaneCisloPaletky = '181' THEN
                i:= 3;
            ELSIF PrecitaneCisloPaletky = '168' THEN
                i:= 4;
            ELSIF PrecitaneCisloPaletky = '140' THEN
                i:= 5;
            ELSIF PrecitaneCisloPaletky = '110' THEN
                i:= 6;
            ELSIF PrecitaneCisloPaletky = '156' THEN
                i:= 7;
            ELSIF PrecitaneCisloPaletky = '127' THEN
                i:= 8;
            ELSIF PrecitaneCisloPaletky = '139' THEN
                i:= 9;
            ELSIF PrecitaneCisloPaletky = '131' THEN
                i:= 10;
            ELSIF PrecitaneCisloPaletky = '178' THEN
                i:= 11;
            ELSIF PrecitaneCisloPaletky = '206' THEN
                i:= 12;
            ELSIF PrecitaneCisloPaletky = '119' THEN
                i:= 13;
            ELSIF PrecitaneCisloPaletky = '163' THEN
                i:= 14;
            ELSIF PrecitaneCisloPaletky = '128' THEN
                i:= 15;
            ELSIF PrecitaneCisloPaletky = '175' THEN
                i:= 16;
            ELSIF PrecitaneCisloPaletky = '138' THEN
                i:= 17;
            ELSE
                P2_Alarmy[214]:= TRUE;
                P2_PoruchaST3:= TRUE;
            END_IF

            IF i<> 0 THEN
                Paletka[i].PAR.CisloPaletky:= USINT_TO_STRING(i);
                P2_StoperSrobovania.PAR.IndexPaletky_STRING:= USINT_TO_STRING(i);
                P2_StoperSrobovania.PAR.IndexPaletky:= i;
                PrecitaneCisloPaletky:= '';
                SC_P2_StoperSrobovania.ResetStep:= TRUE;
                SC_P2_StoperSrobovania.Step:= 104;
            END_IF

        104:
            SC_P2_StoperSrobovania.StepName:='104 - Automaticky Rezim - kontrola stavu paletky';
            SC_P2_StoperSrobovania.IdleTime.PT:= T#200ms;
            SC_P2_StoperSrobovania.AlarmTime.PT:= T#5s;

            IF Paletka[i].PAR.TestovaciKus AND Paletka[i].PAR.CisloTestovacejStanice = 'ST_5' THEN
                TestovaciKus:= TRUE;
            ELSIF Paletka[i].PAR.TestovaciKus AND Paletka[i].PAR.CisloTestovacejStanice <> 'ST_5' THEN
                SC_P2_StoperSrobovania.ResetStep:= TRUE;
                SC_P2_StoperSrobovania.Step:= 560;
            ELSIF Paletka[i].PAR.RevorkovyKus AND Paletka[i].PAR.CisloRevorkovejStanice = 'ST_5' THEN
                Revork:= TRUE;
                SC_P2_StoperSrobovania.ResetStep:= TRUE;
                SC_P2_StoperSrobovania.Step:= 108;
            ELSIF Paletka[i].PAR.RevorkovyKus AND Paletka[i].PAR.CisloRevorkovejStanice <> 'ST_5' THEN
                Revork:= FALSE;
                SC_P2_StoperSrobovania.ResetStep:= TRUE;
                SC_P2_StoperSrobovania.Step:= 560;
            ELSIF Paletka[i].PAR.StavPaletky = 'OK' THEN
                SC_P2_StoperSrobovania.ResetStep:= TRUE;
                SC_P2_StoperSrobovania.Step:= 108;
            ELSIF Paletka[i].PAR.StavPaletky = 'NG' THEN
                SC_P2_StoperSrobovania.ResetStep:= TRUE;
                SC_P2_StoperSrobovania.Step:= 560;
            END_IF

        108:
            SC_P2_StoperSrobovania.StepName:='108 - Automaticky Rezim - vyziadanie stavu paletky zo servera, zacentrovanie paletky';
            SC_P2_StoperSrobovania.IdleTime.PT:= T#200ms;
            SC_P2_StoperSrobovania.AlarmTime.PT:= T#10s;
            SC_P2_StoperSrobovania.IdleTime.IN:= TRUE;

            IF NOT SC_P2_StoperSrobovania.Switch1  THEN
                TRCB_P2_Srobovanie_ST5.CMD.VyziadajStavPaletky_TYP1:= TRUE;
                Centrovacku_VYSUN:= TRUE;
                SC_P2_StoperSrobovania.Switch1:= TRUE;
            END_IF

            IF TRCB_P2_Srobovanie_ST5.STATUS.KomunikaciaUkoncena THEN
                TRCB_P2_Srobovanie_ST5.CMD.VyziadajStavPaletky_TYP1:= FALSE;
                SC_P2_StoperSrobovania.ResetStep:= TRUE;
                SC_P2_StoperSrobovania.Step:= 110;
            ELSIF TRCB_P2_Srobovanie_ST5.STATUS.KomunikaciaError THEN
                TRCB_P2_Srobovanie_ST5.CMD.VyziadajStavPaletky_TYP1:= FALSE;
                SC_P2_StoperSrobovania.ResetStep:= TRUE;
                SC_P2_StoperSrobovania.Step:= 115;
            END_IF

        110:
            SC_P2_StoperSrobovania.StepName:='110 - Automaticky Rezim - kontrola odpovede servera';
            SC_P2_StoperSrobovania.IdleTime.PT:= T#200ms;
            SC_P2_StoperSrobovania.AlarmTime.PT:= T#5s;

            IF NOT TRCB_P2_Srobovanie_ST5.STATUS.KomunikaciaUkoncena AND P2_StoperSrobovania.IN.Centrovanie_VYSUNUTE_IS14 THEN
                IF TRCB_P2_Srobovanie_ST5.OUTPUTS.PovolenieCinnostiNaPaletke = 'OK' THEN
                    Paletka[i].VnutornyStav.KomunikaciaOtvorena:= TRUE;
                    IF TRCB_P2_Srobovanie_ST5.OUTPUTS.DruhCinnostiNaPaletke = 'PRD;ST5' THEN
                        SC_P2_StoperSrobovania.ResetStep:= TRUE;
                        SC_P2_StoperSrobovania.Step:= 118;
                    END_IF
                ELSIF TRCB_P2_Srobovanie_ST5.OUTPUTS.PovolenieCinnostiNaPaletke = 'NG' THEN
                    SC_P2_StoperSrobovania.ResetStep:= TRUE;
                    SC_P2_StoperSrobovania.Step:= 115;
                END_IF
            END_IF

        115:
            SC_P2_StoperSrobovania.StepName:='115 - Automaticky Rezim - rozhodnutie obsluhy po odpovedi panatrace NG';
            SC_P2_StoperSrobovania.IdleTime.PT:= T#200ms;
            SC_P2_StoperSrobovania.AlarmTime.PT:= T#5s;

            P2_Vizu.ZobrazHL4_ST5:= TRUE;

            IF TRCB_P2_Srobov_OpatovnyDopyt THEN
                TRCB_P2_Srobov_OpatovnyDopyt:= FALSE;
                P2_Vizu.ZobrazHL4_ST5:= FALSE;
                SC_P2_StoperSrobovania.ResetStep:= TRUE;
                SC_P2_StoperSrobovania.Step:= 108;
            ELSIF TRCB_P2_Srobov_PaletkaNG THEN
                TRCB_P2_Srobov_PaletkaNG:= FALSE;
                P2_Vizu.ZobrazHL4_ST5:= FALSE;
                Paletka[i].PAR.StavPaletky := 'NG';
                SC_P2_StoperSrobovania.ResetStep:= TRUE;
                SC_P2_StoperSrobovania.Step:= 116;
            END_IF

        116:
            SC_P2_StoperSrobovania.StepName:='116 - Automaticky Rezim - odcentrovanie paletky po odpovedi servera NG';
            SC_P2_StoperSrobovania.IdleTime.PT:= T#200ms;
            SC_P2_StoperSrobovania.AlarmTime.PT:= T#5s;

            IF NOT SC_P2_StoperSrobovania.Switch1 THEN
                Centrovacku_ZASUN:= TRUE;
                SC_P2_StoperSrobovania.Switch1:= TRUE;
            END_IF

            IF P2_StoperSrobovania.IN.Centrovanie_ZASUNUTE_IS15 THEN
                SC_P2_StoperSrobovania.ResetStep:= TRUE;
                SC_P2_StoperSrobovania.Step:= 560;
            END_IF

        118:
            SC_P2_StoperSrobovania.StepName:='118 - Automaticky Rezim - zacentrovanie paletky';
            SC_P2_StoperSrobovania.IdleTime.PT:= T#200ms;
            SC_P2_StoperSrobovania.AlarmTime.PT:= T#5s;

            IF NOT SC_P2_StoperSrobovania.Switch1 THEN
                Centrovacku_VYSUN:= TRUE;
                SC_P2_StoperSrobovania.Switch1:= TRUE;
            END_IF

            IF P2_StoperSrobovania.IN.Centrovanie_VYSUNUTE_IS14 THEN
                SC_P2_StoperSrobovania.ResetStep:= TRUE;
                SC_P2_StoperSrobovania.Step:= 125;
            END_IF

        125:
            SC_P2_StoperSrobovania.StepName:='125 - Automaticky Rezim - rozhodnutie podla typu modelu';
            SC_P2_StoperSrobovania.IdleTime.PT:= T#5s;
            SC_P2_StoperSrobovania.AlarmTime.PT:= T#5s;

            IF Linka.PAR.ZvolenyModel = '4F' THEN
                SC_P2_StoperSrobovania.ResetStep:= TRUE;
                SC_P2_StoperSrobovania.Step:= 138;
            ELSIF Linka.PAR.ZvolenyModel = '5F' THEN
                SC_P2_StoperSrobovania.ResetStep:= TRUE;
                SC_P2_StoperSrobovania.Step:= 258;
            ELSIF Linka.PAR.ZvolenyModel = '5H' THEN
                SC_P2_StoperSrobovania.ResetStep:= TRUE;
                SC_P2_StoperSrobovania.Step:= 358;
            END_IF

            //******************************************Model 4F*************************************************//

        138:
            SC_P2_StoperSrobovania.StepName:='120 - Automaticky Rezim - model 4F presun manipulatora vpred';
            SC_P2_StoperSrobovania.IdleTime.PT:= T#200ms;
            SC_P2_StoperSrobovania.AlarmTime.PT:= T#5s;

            IF NOT SC_P2_StoperSrobovania.Switch1 AND P2_Robot.KOM_IN.Stav_RobotBezpPozicia_Srobovanie THEN
                P2_StoperSrobovania.OUT.KOM_PresunManipulator_DOPREDU:= TRUE;
                SC_P2_StoperSrobovania.Switch1:= TRUE;
            END_IF

            IF P2_Srobovanie.OUT.KOM_PresunVPRED_Ukonceny AND NOT P2_Robot.KOM_IN.Stav_Busbary4F_Odobrate THEN
                P2_Srobovanie.OUT.KOM_PresunVPRED_Ukonceny:= FALSE;
                P2_StoperSrobovania.OUT.KOM_PresunManipulator_DOPREDU:= FALSE;
                SC_P2_StoperSrobovania.ResetStep:= TRUE;
                SC_P2_StoperSrobovania.Step:= 140;
            END_IF

        140:
            SC_P2_StoperSrobovania.StepName:='140 - Automaticky Rezim - modwel 4F odober vrchne busbary';
            SC_P2_StoperSrobovania.IdleTime.PT:= T#200ms;
            SC_P2_StoperSrobovania.AlarmTime.PT:= T#5s;

            P2_Robot.KOM_OUT.ManipSrobovania_BezpecnaPozicia:= TRUE;

            IF NOT SC_P2_StoperSrobovania.Switch1 AND NOT P2_Robot.STAV.Zvaranie_PrebiehaManipulacia THEN
                Paletka[i].VnutornyStav.CinnostSpustena:= TRUE;
                P2_Robot.KOM_OUT.Odober_Busbary4F:= TRUE;
                SC_P2_StoperSrobovania.Switch1:= TRUE;
            END_IF

            IF P2_Robot.KOM_IN.Stav_Busbary4F_Odobrate AND NOT P2_Robot.KOM_IN.Stav_Busbary4F_Polozene THEN
                P2_Robot.KOM_OUT.Odober_Busbary4F:= FALSE;
                SC_P2_StoperSrobovania.ResetStep:= TRUE;
                SC_P2_StoperSrobovania.Step:= 143;
            ELSIF NOT P2_Robot.KOM_IN.Stav_ProgramRUN THEN
                P2_Alarmy[271]:= TRUE;
                P2_PoruchaST3:= TRUE;
            END_IF

        143:
            SC_P2_StoperSrobovania.StepName:='143 - Automaticky Rezim - modwel 4F poloz vrchne busbary';
            SC_P2_StoperSrobovania.IdleTime.PT:= T#200ms;
            SC_P2_StoperSrobovania.AlarmTime.PT:= T#5s;

            P2_Robot.KOM_OUT.ManipSrobovania_BezpecnaPozicia:= TRUE;

            IF NOT SC_P2_StoperSrobovania.Switch1 THEN
                P2_Robot.KOM_OUT.Poloz_Busbary4F:= TRUE;
                SC_P2_StoperSrobovania.Switch1:= TRUE;
            END_IF

            IF P2_Robot.KOM_IN.Stav_Busbary4F_Polozene THEN
                P2_Robot.KOM_OUT.Poloz_Busbary4F:= FALSE;
                SC_P2_StoperSrobovania.ResetStep:= TRUE;
                SC_P2_StoperSrobovania.Step:= 145;
            ELSIF NOT P2_Robot.KOM_IN.Stav_ProgramRUN THEN
                P2_Alarmy[271]:= TRUE;
                P2_PoruchaST3:= TRUE;
            END_IF

        145:
            SC_P2_StoperSrobovania.StepName:='145 - Automaticky Rezim - modwel 4F zaskrutkuj lavu skrutku M6';
            SC_P2_StoperSrobovania.IdleTime.PT:= T#200ms;
            SC_P2_StoperSrobovania.AlarmTime.PT:= T#5s;

            IF NOT SC_P2_StoperSrobovania.Switch1 THEN
                P2_Srobovanie.STAV.Vysledok_Srobovania:= '';
                P2_StoperSrobovania.OUT.KOM_4F_ZasrobujLavuSkrutkuM6:= TRUE;
                SC_P2_StoperSrobovania.Switch1:= TRUE;
            END_IF

            IF P2_Srobovanie.OUT.KOM_Srobovanie_Ukoncene THEN
                P2_Srobovanie.OUT.KOM_Srobovanie_Ukoncene:= FALSE;
                P2_StoperSrobovania.OUT.KOM_4F_ZasrobujLavuSkrutkuM6:= FALSE;
                IF P2_StoperSrobovania.STAV.Porucha THEN
                    SC_P2_StoperSrobovania.ResetStep:= TRUE;
                    SC_P2_StoperSrobovania.Step:= 500;
                ELSE
                    SC_P2_StoperSrobovania.ResetStep:= TRUE;
                    SC_P2_StoperSrobovania.Step:= 148;
                END_IF
            END_IF

        148:
            SC_P2_StoperSrobovania.StepName:='148 - Automaticky Rezim - modwel 4F kontrola vysledku zaskrutkovania lavej skrutky M6';
            SC_P2_StoperSrobovania.IdleTime.PT:= T#200ms;
            SC_P2_StoperSrobovania.AlarmTime.PT:= T#5s;

            Reports.Skrutkovacky.Moment_ToleranciaMIN.P2_LavaSkrutkaM6:= REAL_TO_STRING(P2_Srobovanie.STAV.M6_Moment_ToleranciaMIN_REAL);
            Reports.Skrutkovacky.Moment_ToleranciaMAX.P2_LavaSkrutkaM6:= REAL_TO_STRING(P2_Srobovanie.STAV.M6_Moment_ToleranciaMAX_REAL);
            Reports.Skrutkovacky.Moment_NameranaHodnota.P2_LavaSkrutkaM6:= REAL_TO_STRING(P2_Srobovanie.STAV.M6_DosiahnutyMoment_REAL);
            Reports.Skrutkovacky.Uhol_ToleranciaMIN.P2_LavaSkrutkaM6:= UDINT_TO_STRING(P2_Srobovanie.STAV.M6_Uhol_ToleranciaMIN);
            Reports.Skrutkovacky.Uhol_ToleranciaMAX.P2_LavaSkrutkaM6:= UDINT_TO_STRING(P2_Srobovanie.STAV.M6_Uhol_ToleranciaMAX);
            Reports.Skrutkovacky.Uhol_NameranaHodnota.P2_LavaSkrutkaM6:= UDINT_TO_STRING(P2_Srobovanie.STAV.M6_DosiahnutyUhol);

            IF NOT SC_P2_StoperSrobovania.Switch1 THEN
                P2_Skrutk_4F_LavaM6_Vysunutie:= STRING_TO_REAL(Reports.Skrutkovacky.VyskaSkrutkovania.P2_LavaSkrutkaM6);
                IF (P2_Skrutk_4F_LavaM6_Vysunutie <= P2_RemPremenne.P2_Srob4F_LavaM6_Vysunutie_HI) AND (P2_Skrutk_4F_LavaM6_Vysunutie >= P2_RemPremenne.P2_Srob4F_LavaM6_Vysunutie_LO)THEN
                    VysunutieSkrutkovacky_OK:= TRUE;
                ELSE
                    VysunutieSkrutkovacky_OK:= FALSE;
                END_IF
                SC_P2_StoperSrobovania.Switch1:= TRUE;
            END_IF

            IF P2_Srobovanie.STAV.Vysledok_Srobovania = 'OK' THEN
                IF VysunutieSkrutkovacky_OK THEN
                    Reports.Skrutkovacky.VyslednyReport.P2_LavaSkrutkaM6:= 'PASS';
                    SC_P2_StoperSrobovania.ResetStep:= TRUE;
                    SC_P2_StoperSrobovania.Step:= 150;
                ELSE
                    Reports.Skrutkovacky.VyslednyReport.P2_LavaSkrutkaM6:= 'FAIL';
                    IF P2_Srobov_M6_Result_OFF THEN
                        SC_P2_StoperSrobovania.ResetStep:= TRUE;
                        SC_P2_StoperSrobovania.Step:= 150;
                    ELSE
                        SC_P2_StoperSrobovania.ResetStep:= TRUE;
                        SC_P2_StoperSrobovania.Step:= 500;
                    END_IF
                END_IF
            ELSIF P2_Srobovanie.STAV.Vysledok_Srobovania = 'NG' THEN
                Reports.Skrutkovacky.VyslednyReport.P2_LavaSkrutkaM6:= 'FAIL';
                IF P2_Srobov_M6_Result_OFF THEN
                    SC_P2_StoperSrobovania.ResetStep:= TRUE;
                    SC_P2_StoperSrobovania.Step:= 150;
                ELSE
                    SC_P2_StoperSrobovania.ResetStep:= TRUE;
                    SC_P2_StoperSrobovania.Step:= 500;
                END_IF
            END_IF

        150:
            SC_P2_StoperSrobovania.StepName:='150 - Automaticky Rezim - modwel 4F zaskrutkuj pravu skrutku M6';
            SC_P2_StoperSrobovania.IdleTime.PT:= T#200ms;
            SC_P2_StoperSrobovania.AlarmTime.PT:= T#5s;

            IF NOT SC_P2_StoperSrobovania.Switch1 THEN
                P2_Srobovanie.STAV.Vysledok_Srobovania:= '';
                P2_StoperSrobovania.OUT.KOM_4F_ZasrobujPravuSkrutkuM6:= TRUE;
                SC_P2_StoperSrobovania.Switch1:= TRUE;
            END_IF

            IF P2_Srobovanie.OUT.KOM_Srobovanie_Ukoncene THEN
                P2_Srobovanie.OUT.KOM_Srobovanie_Ukoncene:= FALSE;
                P2_StoperSrobovania.OUT.KOM_4F_ZasrobujPravuSkrutkuM6:= FALSE;
                IF P2_StoperSrobovania.STAV.Porucha THEN
                    SC_P2_StoperSrobovania.ResetStep:= TRUE;
                    SC_P2_StoperSrobovania.Step:= 500;
                ELSE
                    SC_P2_StoperSrobovania.ResetStep:= TRUE;
                    SC_P2_StoperSrobovania.Step:= 153;
                END_IF
            END_IF

        153:
            SC_P2_StoperSrobovania.StepName:='151 - Automaticky Rezim - modwel 4F kontrola vysledku zaskrutkovania pravej skrutky M6';
            SC_P2_StoperSrobovania.IdleTime.PT:= T#200ms;
            SC_P2_StoperSrobovania.AlarmTime.PT:= T#5s;

            Reports.Skrutkovacky.Moment_ToleranciaMIN.P2_PravaSkrutkaM6:= REAL_TO_STRING(P2_Srobovanie.STAV.M6_Moment_ToleranciaMIN_REAL);
            Reports.Skrutkovacky.Moment_ToleranciaMAX.P2_PravaSkrutkaM6:= REAL_TO_STRING(P2_Srobovanie.STAV.M6_Moment_ToleranciaMAX_REAL);
            Reports.Skrutkovacky.Moment_NameranaHodnota.P2_PravaSkrutkaM6:= REAL_TO_STRING(P2_Srobovanie.STAV.M6_DosiahnutyMoment_REAL);
            Reports.Skrutkovacky.Uhol_ToleranciaMIN.P2_PravaSkrutkaM6:= UDINT_TO_STRING(P2_Srobovanie.STAV.M6_Uhol_ToleranciaMIN);
            Reports.Skrutkovacky.Uhol_ToleranciaMAX.P2_PravaSkrutkaM6:= UDINT_TO_STRING(P2_Srobovanie.STAV.M6_Uhol_ToleranciaMAX);
            Reports.Skrutkovacky.Uhol_NameranaHodnota.P2_PravaSkrutkaM6:= UDINT_TO_STRING(P2_Srobovanie.STAV.M6_DosiahnutyUhol);

            IF NOT SC_P2_StoperSrobovania.Switch1 THEN
                P2_Skrutk_4F_PravaM6_Vysunutie:= STRING_TO_REAL(Reports.Skrutkovacky.VyskaSkrutkovania.P2_PravaSkrutkaM6);
                IF (P2_Skrutk_4F_PravaM6_Vysunutie <= P2_RemPremenne.P2_Srob4F_PravaM6_Vysunutie_HI) AND (P2_Skrutk_4F_PravaM6_Vysunutie >= P2_RemPremenne.P2_Srob4F_PravaM6_Vysunutie_LO)THEN
                    VysunutieSkrutkovacky_OK:= TRUE;
                ELSE
                    VysunutieSkrutkovacky_OK:= FALSE;
                END_IF
                SC_P2_StoperSrobovania.Switch1:= TRUE;
            END_IF

            IF P2_Srobovanie.STAV.Vysledok_Srobovania = 'OK' THEN
                IF VysunutieSkrutkovacky_OK THEN
                    Reports.Skrutkovacky.VyslednyReport.P2_PravaSkrutkaM6:= 'PASS';
                    SC_P2_StoperSrobovania.ResetStep:= TRUE;
                    SC_P2_StoperSrobovania.Step:= 155;
                ELSE
                    Reports.Skrutkovacky.VyslednyReport.P2_PravaSkrutkaM6:= 'FAIL';
                    IF P2_Srobov_M6_Result_OFF THEN
                        SC_P2_StoperSrobovania.ResetStep:= TRUE;
                        SC_P2_StoperSrobovania.Step:= 155;
                    ELSE
                        SC_P2_StoperSrobovania.ResetStep:= TRUE;
                        SC_P2_StoperSrobovania.Step:= 500;
                    END_IF
                END_IF
            ELSIF P2_Srobovanie.STAV.Vysledok_Srobovania = 'NG' THEN
                Reports.Skrutkovacky.VyslednyReport.P2_PravaSkrutkaM6:= 'FAIL';
                IF P2_Srobov_M6_Result_OFF THEN
                    SC_P2_StoperSrobovania.ResetStep:= TRUE;
                    SC_P2_StoperSrobovania.Step:= 155;
                ELSE
                    SC_P2_StoperSrobovania.ResetStep:= TRUE;
                    SC_P2_StoperSrobovania.Step:= 500;
                END_IF
            END_IF

        155:
            SC_P2_StoperSrobovania.StepName:='155 - Automaticky Rezim - modwel 4F presun manipulatora vpred';
            SC_P2_StoperSrobovania.IdleTime.PT:= T#200ms;
            SC_P2_StoperSrobovania.AlarmTime.PT:= T#5s;

            IF NOT SC_P2_StoperSrobovania.Switch1 THEN
                P2_StoperSrobovania.OUT.KOM_PresunManipulator_DOPREDU:= TRUE;
                SC_P2_StoperSrobovania.Switch1:= TRUE;
            END_IF

            IF P2_Srobovanie.OUT.KOM_PresunVPRED_Ukonceny AND NOT P2_Robot.KOM_IN.Stav_RobotPoziciaCakania THEN
                P2_Srobovanie.OUT.KOM_PresunVPRED_Ukonceny:= FALSE;
                P2_StoperSrobovania.OUT.KOM_PresunManipulator_DOPREDU:= FALSE;
                SC_P2_StoperSrobovania.ResetStep:= TRUE;
                SC_P2_StoperSrobovania.Step:= 158;
            END_IF

        158:
            SC_P2_StoperSrobovania.StepName:='158 - Automaticky Rezim - model 4F vystavenie signalu pre robota chod do cakacej pozicie';
            SC_P2_StoperSrobovania.IdleTime.PT:= T#200ms;
            SC_P2_StoperSrobovania.AlarmTime.PT:= T#5s;

            P2_Robot.KOM_OUT.ManipSrobovania_BezpecnaPozicia:= TRUE;

            IF NOT SC_P2_StoperSrobovania.Switch1 THEN
                P2_Robot.KOM_OUT.Presun_CakaciaPozicia:= TRUE;
                SC_P2_StoperSrobovania.Switch1:= TRUE;
            END_IF

            IF P2_Robot.KOM_IN.Stav_RobotPoziciaCakania THEN
                P2_Robot.STAV.Srobovanie_PrebiehaManipulacia:= FALSE;
                P2_Robot.KOM_OUT.Presun_CakaciaPozicia:= FALSE;
                SC_P2_StoperSrobovania.ResetStep:= TRUE;
                SC_P2_StoperSrobovania.Step:= 160;
            END_IF

        160:
            SC_P2_StoperSrobovania.StepName:='160 - Automaticky Rezim - modwel 4F zaskrutkuj lavu skrutku M4';
            SC_P2_StoperSrobovania.IdleTime.PT:= T#200ms;
            SC_P2_StoperSrobovania.AlarmTime.PT:= T#5s;

            IF NOT SC_P2_StoperSrobovania.Switch1 AND P2_Robot.KOM_IN.Stav_RobotBezpPozicia_Srobovanie THEN
                P2_Srobovanie.STAV.Vysledok_Srobovania:= '';
                P2_StoperSrobovania.OUT.KOM_4F_ZasrobujLavuSkrutkuM4:= TRUE;
                SC_P2_StoperSrobovania.Switch1:= TRUE;
            END_IF

            IF P2_Srobovanie.OUT.KOM_Srobovanie_Ukoncene THEN
                P2_Srobovanie.OUT.KOM_Srobovanie_Ukoncene:= FALSE;
                P2_StoperSrobovania.OUT.KOM_4F_ZasrobujLavuSkrutkuM4:= FALSE;
                IF P2_StoperSrobovania.STAV.Porucha THEN
                    SC_P2_StoperSrobovania.ResetStep:= TRUE;
                    SC_P2_StoperSrobovania.Step:= 500;
                ELSE
                    SC_P2_StoperSrobovania.ResetStep:= TRUE;
                    SC_P2_StoperSrobovania.Step:= 163;
                END_IF
            END_IF

        163:
            SC_P2_StoperSrobovania.StepName:='163 - Automaticky Rezim - modwel 4F kontrola vysledku zaskrutkovania lavej skrutky M4';
            SC_P2_StoperSrobovania.IdleTime.PT:= T#200ms;
            SC_P2_StoperSrobovania.AlarmTime.PT:= T#5s;

            Reports.Skrutkovacky.Moment_ToleranciaMIN.P2_LavaSkrutkaM4:= REAL_TO_STRING(P2_Srobovanie.STAV.M4_Moment_ToleranciaMIN_REAL);
            Reports.Skrutkovacky.Moment_ToleranciaMAX.P2_LavaSkrutkaM4:= REAL_TO_STRING(P2_Srobovanie.STAV.M4_Moment_ToleranciaMAX_REAL);
            Reports.Skrutkovacky.Moment_NameranaHodnota.P2_LavaSkrutkaM4:= REAL_TO_STRING(P2_Srobovanie.STAV.M4_DosiahnutyMoment_REAL);
            Reports.Skrutkovacky.Uhol_ToleranciaMIN.P2_LavaSkrutkaM4:= UDINT_TO_STRING(P2_Srobovanie.STAV.M4_Uhol_ToleranciaMIN);
            Reports.Skrutkovacky.Uhol_ToleranciaMAX.P2_LavaSkrutkaM4:= UDINT_TO_STRING(P2_Srobovanie.STAV.M4_Uhol_ToleranciaMAX);
            Reports.Skrutkovacky.Uhol_NameranaHodnota.P2_LavaSkrutkaM4:= UDINT_TO_STRING(P2_Srobovanie.STAV.M4_DosiahnutyUhol);

            IF NOT SC_P2_StoperSrobovania.Switch1 THEN
                P2_Skrutk_4F_LavaM4_Vysunutie:= STRING_TO_REAL(Reports.Skrutkovacky.VyskaSkrutkovania.P2_LavaSkrutkaM4);
                IF (P2_Skrutk_4F_LavaM4_Vysunutie <= P2_RemPremenne.P2_Srob4F_LavaM4_Vysunutie_HI) AND (P2_Skrutk_4F_LavaM4_Vysunutie >= P2_RemPremenne.P2_Srob4F_LavaM4_Vysunutie_LO)THEN
                    VysunutieSkrutkovacky_OK:= TRUE;
                ELSE
                    VysunutieSkrutkovacky_OK:= FALSE;
                END_IF
                SC_P2_StoperSrobovania.Switch1:= TRUE;
            END_IF

            IF P2_Srobovanie.STAV.Vysledok_Srobovania = 'OK' THEN
                IF VysunutieSkrutkovacky_OK THEN
                    Reports.Skrutkovacky.VyslednyReport.P2_LavaSkrutkaM4:= 'PASS';
                    SC_P2_StoperSrobovania.ResetStep:= TRUE;
                    SC_P2_StoperSrobovania.Step:= 165;
                ELSE
                    Reports.Skrutkovacky.VyslednyReport.P2_LavaSkrutkaM4:= 'FAIL';
                    IF P2_Srobov_M4_Result_OFF THEN
                        SC_P2_StoperSrobovania.ResetStep:= TRUE;
                        SC_P2_StoperSrobovania.Step:= 165;
                    ELSE
                        SC_P2_StoperSrobovania.ResetStep:= TRUE;
                        SC_P2_StoperSrobovania.Step:= 500;
                    END_IF
                END_IF
            ELSIF P2_Srobovanie.STAV.Vysledok_Srobovania = 'NG' THEN
                Reports.Skrutkovacky.VyslednyReport.P2_LavaSkrutkaM4:= 'FAIL';
                IF P2_Srobov_M4_Result_OFF THEN
                    SC_P2_StoperSrobovania.ResetStep:= TRUE;
                    SC_P2_StoperSrobovania.Step:= 165;
                ELSE
                    SC_P2_StoperSrobovania.ResetStep:= TRUE;
                    SC_P2_StoperSrobovania.Step:= 500;
                END_IF
            END_IF

        165:
            SC_P2_StoperSrobovania.StepName:='165 - Automaticky Rezim - modwel 4F zaskrutkuj pravu skrutku M4';
            SC_P2_StoperSrobovania.IdleTime.PT:= T#200ms;
            SC_P2_StoperSrobovania.AlarmTime.PT:= T#5s;

            IF NOT SC_P2_StoperSrobovania.Switch1 AND P2_Robot.KOM_IN.Stav_RobotBezpPozicia_Srobovanie THEN
                P2_Srobovanie.STAV.Vysledok_Srobovania:= '';
                P2_StoperSrobovania.OUT.KOM_4F_ZasrobujPravuSkrutkuM4:= TRUE;
                SC_P2_StoperSrobovania.Switch1:= TRUE;
            END_IF

            IF P2_Srobovanie.OUT.KOM_Srobovanie_Ukoncene THEN
                P2_Srobovanie.OUT.KOM_Srobovanie_Ukoncene:= FALSE;
                P2_StoperSrobovania.OUT.KOM_4F_ZasrobujPravuSkrutkuM4:= FALSE;
                IF P2_StoperSrobovania.STAV.Porucha THEN
                    SC_P2_StoperSrobovania.ResetStep:= TRUE;
                    SC_P2_StoperSrobovania.Step:= 500;
                ELSE
                    SC_P2_StoperSrobovania.ResetStep:= TRUE;
                    SC_P2_StoperSrobovania.Step:= 168;
                END_IF
            END_IF

        168:
            SC_P2_StoperSrobovania.StepName:='168 - Automaticky Rezim - modwel 4F kontrola vysledku zaskrutkovania pravej skrutky M4';
            SC_P2_StoperSrobovania.IdleTime.PT:= T#200ms;
            SC_P2_StoperSrobovania.AlarmTime.PT:= T#5s;

            Reports.Skrutkovacky.Moment_ToleranciaMIN.P2_PravaSkrutkaM4:= REAL_TO_STRING(P2_Srobovanie.STAV.M4_Moment_ToleranciaMIN_REAL);
            Reports.Skrutkovacky.Moment_ToleranciaMAX.P2_PravaSkrutkaM4:= REAL_TO_STRING(P2_Srobovanie.STAV.M4_Moment_ToleranciaMAX_REAL);
            Reports.Skrutkovacky.Moment_NameranaHodnota.P2_PravaSkrutkaM4:= REAL_TO_STRING(P2_Srobovanie.STAV.M4_DosiahnutyMoment_REAL);
            Reports.Skrutkovacky.Uhol_ToleranciaMIN.P2_PravaSkrutkaM4:= UDINT_TO_STRING(P2_Srobovanie.STAV.M4_Uhol_ToleranciaMIN);
            Reports.Skrutkovacky.Uhol_ToleranciaMAX.P2_PravaSkrutkaM4:= UDINT_TO_STRING(P2_Srobovanie.STAV.M4_Uhol_ToleranciaMAX);
            Reports.Skrutkovacky.Uhol_NameranaHodnota.P2_PravaSkrutkaM4:= UDINT_TO_STRING(P2_Srobovanie.STAV.M4_DosiahnutyUhol);

            IF NOT SC_P2_StoperSrobovania.Switch1 THEN
                P2_Skrutk_4F_PravaM4_Vysunutie:= STRING_TO_REAL(Reports.Skrutkovacky.VyskaSkrutkovania.P2_PravaSkrutkaM4);
                IF (P2_Skrutk_4F_PravaM4_Vysunutie <= P2_RemPremenne.P2_Srob4F_PravaM4_Vysunutie_HI) AND (P2_Skrutk_4F_PravaM4_Vysunutie >= P2_RemPremenne.P2_Srob4F_PravaM4_Vysunutie_LO)THEN
                    VysunutieSkrutkovacky_OK:= TRUE;
                ELSE
                    VysunutieSkrutkovacky_OK:= FALSE;
                END_IF
                SC_P2_StoperSrobovania.Switch1:= TRUE;
            END_IF

            IF P2_Srobovanie.STAV.Vysledok_Srobovania = 'OK' THEN
                IF VysunutieSkrutkovacky_OK THEN
                    Reports.Skrutkovacky.VyslednyReport.P2_PravaSkrutkaM4:= 'PASS';
                    SC_P2_StoperSrobovania.ResetStep:= TRUE;
                    SC_P2_StoperSrobovania.Step:= 170;
                ELSE
                    Reports.Skrutkovacky.VyslednyReport.P2_PravaSkrutkaM4:= 'FAIL';
                    IF P2_Srobov_M4_Result_OFF THEN
                        SC_P2_StoperSrobovania.ResetStep:= TRUE;
                        SC_P2_StoperSrobovania.Step:= 170;
                    ELSE
                        SC_P2_StoperSrobovania.ResetStep:= TRUE;
                        SC_P2_StoperSrobovania.Step:= 500;
                    END_IF
                END_IF
            ELSIF P2_Srobovanie.STAV.Vysledok_Srobovania = 'NG' THEN
                Reports.Skrutkovacky.VyslednyReport.P2_PravaSkrutkaM4:= 'FAIL';
                IF P2_Srobov_M4_Result_OFF THEN
                    SC_P2_StoperSrobovania.ResetStep:= TRUE;
                    SC_P2_StoperSrobovania.Step:= 170;
                ELSE
                    SC_P2_StoperSrobovania.ResetStep:= TRUE;
                    SC_P2_StoperSrobovania.Step:= 500;
                END_IF
            END_IF

        170:
            SC_P2_StoperSrobovania.StepName:='170 - Automaticky Rezim - modwel 4F presun manipulatora vzad';
            SC_P2_StoperSrobovania.IdleTime.PT:= T#200ms;
            SC_P2_StoperSrobovania.AlarmTime.PT:= T#5s;

            IF NOT SC_P2_StoperSrobovania.Switch1 AND P2_Robot.KOM_IN.Stav_RobotBezpPozicia_Srobovanie THEN
                P2_StoperSrobovania.OUT.KOM_PresunManipulator_DOZADU:= TRUE;
                SC_P2_StoperSrobovania.Switch1:= TRUE;
            END_IF

            IF P2_Srobovanie.OUT.KOM_PresunVZAD_Ukonceny THEN
                P2_Srobovanie.OUT.KOM_PresunVZAD_Ukonceny:= FALSE;
                P2_StoperSrobovania.OUT.KOM_PresunManipulator_DOZADU:= FALSE;
                CAM10.STAV.Results_READY:= FALSE;
                SC_P2_StoperSrobovania.ResetStep:= TRUE;
                SC_P2_StoperSrobovania.Step:= 173;
            END_IF

        173:
            SC_P2_StoperSrobovania.StepName:='173 - Automaticky Rezim - modwel 4F kamerova kontrola paletky CAM10';//CAM 10//
            SC_P2_StoperSrobovania.IdleTime.PT:= T#5s;
            SC_P2_StoperSrobovania.AlarmTime.PT:= T#5s;

            IF NOT SC_P2_StoperSrobovania.Switch1 AND CAM10.STAV.Command_READY THEN
                CAM10.CMD.Triger:= TRUE;
                SC_P2_StoperSrobovania.IdleTime.IN:= TRUE;
                SC_P2_StoperSrobovania.Switch1:= TRUE;
            END_IF

            IF CAM10.STAV.Results_READY AND CAM10.STAV.Command_AKCEPTOVANY THEN
                PocetTrigrovKamery:= 0;
                CAM10.STAV.Results_READY:= FALSE;
                SC_P2_StoperSrobovania.ResetStep:= TRUE;
                SC_P2_StoperSrobovania.Step:= 175;
            ELSIF SC_P2_StoperSrobovania.IdleTime.Q AND PocetTrigrovKamery < 5 THEN
                PocetTrigrovKamery:= PocetTrigrovKamery + 1;
                CAM10.STAV.Results_READY:= FALSE;
                CAM10.CMD.Triger:= FALSE;
                SC_P2_StoperSrobovania.ResetStep:= TRUE;
                SC_P2_StoperSrobovania.Step:= 174;
            ELSIF SC_P2_StoperSrobovania.IdleTime.Q AND PocetTrigrovKamery >= 5 THEN
                P2_Alarmy[295]:= TRUE;
                P2_PoruchaST3:= TRUE;
            END_IF

        174:
            SC_P2_StoperSrobovania.StepName:='174 - Automaticky Rezim - modwel 4F cakam na opatovny triger kamery';//CAM 10//
            SC_P2_StoperSrobovania.IdleTime.PT:= T#1s;
            SC_P2_StoperSrobovania.AlarmTime.PT:= T#5s;

            SC_P2_StoperSrobovania.IdleTime.IN:= TRUE;

            IF SC_P2_StoperSrobovania.IdleTime.Q THEN
                SC_P2_StoperSrobovania.ResetStep:= TRUE;
                SC_P2_StoperSrobovania.Step:= 173;
            END_IF

        175:
            SC_P2_StoperSrobovania.StepName:='175 - Automaticky Rezim - model 4F kontrola vysledku kamery';
            SC_P2_StoperSrobovania.IdleTime.PT:= T#200ms;
            SC_P2_StoperSrobovania.AlarmTime.PT:= T#5s;
            SC_P2_StoperSrobovania.IdleTime.IN:= TRUE;

            IF NOT CAM10.STAV.BUSY THEN
                CAM10.CMD.Triger:= FALSE;
                IF NOT CAM10.RESULT.Paletka.Pritomn_Busbarov_4F	THEN
					CAM10.PAR.ResultFotky:= 'PASS';
					SC_P2_StoperSrobovania.ResetStep:= TRUE;
					SC_P2_StoperSrobovania.Step:= 180;
                ELSE
                    CAM10.PAR.ResultFotky:= 'FAIL';
                    SC_P2_StoperSrobovania.ResetStep:= TRUE;
                    SC_P2_StoperSrobovania.Step:= 180;
                END_IF
            END_IF

        180:
            SC_P2_StoperSrobovania.StepName:='135 - Automaticky Rezim - model 4F rozhodnutie podla kamerovej kontroly paletky';
            SC_P2_StoperSrobovania.IdleTime.PT:= T#200ms;
            SC_P2_StoperSrobovania.AlarmTime.PT:= T#5s;
            P2_Srobov_CakaNaKameru:= TRUE;

            IF CAM10.PAR.ResultFotky = 'PASS' THEN
                Paletka[i].VnutornyStav.CinnostUkoncena:= TRUE;
                Paletka[i].PAR.StavPowerCP:= 'PASS';
                P2_Srobov_CakaNaKameru:= FALSE;
                SC_P2_StoperSrobovania.ResetStep:= TRUE;
                SC_P2_StoperSrobovania.Step:= 540;
            ELSIF CAM10.PAR.ResultFotky = 'FAIL' THEN
                P2_Vizu.ZobrazHL1_ST5:= TRUE;
                Paletka[i].VnutornyStav.CinnostUkoncena:= TRUE;
                IF P2_Srobov_KAM_Result_OFF THEN
                    Paletka[i].PAR.StavPowerCP:= 'PASS';
                    P2_Vizu.ZobrazHL1_ST5:= FALSE;
                    P2_Srobov_CakaNaKameru:= FALSE;
                    SC_P2_StoperSrobovania.ResetStep:= TRUE;
                    SC_P2_StoperSrobovania.Step:= 540;
                ELSIF P2_Srobov_KAM_Result_OK THEN
                    P2_Srobov_KAM_Result_OK:= FALSE;
                    Paletka[i].PAR.StavPowerCP:= 'PASS';
                    CAM10.PAR.ResultFotky:= 'PASS';
                    P2_Vizu.ZobrazHL1_ST5:= FALSE;
                    P2_Srobov_CakaNaKameru:= FALSE;
                    SC_P2_StoperSrobovania.ResetStep:= TRUE;
                    SC_P2_StoperSrobovania.Step:= 540;
                ELSIF P2_Srobov_KAM_Result_NG THEN
                    P2_Srobov_KAM_Result_NG:= FALSE;
                    P2_Vizu.ZobrazHL1_ST5:= FALSE;
                    Paletka[i].PAR.StavPowerCP:= 'FAIL';
                    P2_Srobov_CakaNaKameru:= FALSE;
                    SC_P2_StoperSrobovania.ResetStep:= TRUE;
                    SC_P2_StoperSrobovania.Step:= 540;
                END_IF
            END_IF

            //********************************************Model 5F**************************************************************//

        258:
            SC_P2_StoperSrobovania.StepName:='120 - Automaticky Rezim - model 5F presun manipulatora vpred';
            SC_P2_StoperSrobovania.IdleTime.PT:= T#200ms;
            SC_P2_StoperSrobovania.AlarmTime.PT:= T#5s;

            IF NOT SC_P2_StoperSrobovania.Switch1 AND P2_Robot.KOM_IN.Stav_RobotBezpPozicia_Srobovanie THEN
                P2_StoperSrobovania.OUT.KOM_PresunManipulator_DOPREDU:= TRUE;
                SC_P2_StoperSrobovania.Switch1:= TRUE;
            END_IF

            IF P2_Srobovanie.STAV.OsY_AktualnaPozicia > 250 THEN
                P2_Robot.KOM_OUT.ManipSrobovania_BezpecnaPozicia:= TRUE;
                P2_Robot.KOM_OUT.Odober_Busbary5F:= TRUE;
            END_IF

            IF P2_Srobovanie.OUT.KOM_PresunVPRED_Ukonceny AND NOT P2_Robot.KOM_IN.Stav_Busbary5F_Odobrate THEN
                P2_Srobovanie.OUT.KOM_PresunVPRED_Ukonceny:= FALSE;
                P2_StoperSrobovania.OUT.KOM_PresunManipulator_DOPREDU:= FALSE;
                SC_P2_StoperSrobovania.ResetStep:= TRUE;
                SC_P2_StoperSrobovania.Step:= 260;
            END_IF

        260:
            SC_P2_StoperSrobovania.StepName:='260 - Automaticky Rezim - modwel 5F odober vrchne busbary';
            SC_P2_StoperSrobovania.IdleTime.PT:= T#200ms;
            SC_P2_StoperSrobovania.AlarmTime.PT:= T#5s;

            P2_Robot.KOM_OUT.ManipSrobovania_BezpecnaPozicia:= TRUE;

            IF NOT SC_P2_StoperSrobovania.Switch1 AND NOT P2_Robot.STAV.Zvaranie_PrebiehaManipulacia THEN
                Paletka[i].VnutornyStav.CinnostSpustena:= TRUE;
                P2_Robot.KOM_OUT.Odober_Busbary5F:= TRUE;
                SC_P2_StoperSrobovania.Switch1:= TRUE;
            END_IF

            IF P2_Robot.KOM_IN.Stav_Busbary5F_Odobrate AND NOT P2_Robot.KOM_IN.Stav_Busbary5F_Polozene THEN
                P2_Robot.KOM_OUT.Odober_Busbary5F:= FALSE;
                SC_P2_StoperSrobovania.ResetStep:= TRUE;
                SC_P2_StoperSrobovania.Step:= 263;
            ELSIF NOT P2_Robot.KOM_IN.Stav_ProgramRUN THEN
                P2_Alarmy[271]:= TRUE;
                P2_PoruchaST3:= TRUE;
            END_IF

        263:
            SC_P2_StoperSrobovania.StepName:='263 - Automaticky Rezim - modwel 5F poloz vrchne busbary';
            SC_P2_StoperSrobovania.IdleTime.PT:= T#200ms;
            SC_P2_StoperSrobovania.AlarmTime.PT:= T#5s;

            P2_Robot.KOM_OUT.ManipSrobovania_BezpecnaPozicia:= TRUE;

            IF NOT SC_P2_StoperSrobovania.Switch1 THEN
                P2_Robot.KOM_OUT.Poloz_Busbary5F:= TRUE;
                SC_P2_StoperSrobovania.Switch1:= TRUE;
            END_IF

            IF P2_Robot.KOM_IN.Stav_Busbary5F_Polozene THEN
                P2_Robot.KOM_OUT.Poloz_Busbary5F:= FALSE;
                SC_P2_StoperSrobovania.ResetStep:= TRUE;
                SC_P2_StoperSrobovania.Step:= 265;
            ELSIF NOT P2_Robot.KOM_IN.Stav_ProgramRUN THEN
                P2_Alarmy[271]:= TRUE;
                P2_PoruchaST3:= TRUE;
            END_IF

        265:
            SC_P2_StoperSrobovania.StepName:='265 - Automaticky Rezim - modwel 5F zaskrutkuj lavu skrutku M6';
            SC_P2_StoperSrobovania.IdleTime.PT:= T#200ms;
            SC_P2_StoperSrobovania.AlarmTime.PT:= T#5s;

            IF NOT SC_P2_StoperSrobovania.Switch1 THEN
                P2_Srobovanie.STAV.Vysledok_Srobovania:= '';
                P2_StoperSrobovania.OUT.KOM_5F_ZasrobujLavuSkrutkuM6:= TRUE;
                SC_P2_StoperSrobovania.Switch1:= TRUE;
            END_IF

            IF P2_Srobovanie.OUT.KOM_Srobovanie_Ukoncene THEN
                P2_Srobovanie.OUT.KOM_Srobovanie_Ukoncene:= FALSE;
                P2_StoperSrobovania.OUT.KOM_5F_ZasrobujLavuSkrutkuM6:= FALSE;
                IF P2_StoperSrobovania.STAV.Porucha THEN
                    SC_P2_StoperSrobovania.ResetStep:= TRUE;
                    SC_P2_StoperSrobovania.Step:= 500;
                ELSE
                    SC_P2_StoperSrobovania.ResetStep:= TRUE;
                    SC_P2_StoperSrobovania.Step:= 268;
                END_IF
            END_IF

        268:
            SC_P2_StoperSrobovania.StepName:='268 - Automaticky Rezim - modwel 5F kontrola vysledku zaskrutkovania lavej skrutky M6';
            SC_P2_StoperSrobovania.IdleTime.PT:= T#200ms;
            SC_P2_StoperSrobovania.AlarmTime.PT:= T#5s;

            Reports.Skrutkovacky.Moment_ToleranciaMIN.P2_LavaSkrutkaM6:= REAL_TO_STRING(P2_Srobovanie.STAV.M6_Moment_ToleranciaMIN_REAL);
            Reports.Skrutkovacky.Moment_ToleranciaMAX.P2_LavaSkrutkaM6:= REAL_TO_STRING(P2_Srobovanie.STAV.M6_Moment_ToleranciaMAX_REAL);
            Reports.Skrutkovacky.Moment_NameranaHodnota.P2_LavaSkrutkaM6:= REAL_TO_STRING(P2_Srobovanie.STAV.M6_DosiahnutyMoment_REAL);
            Reports.Skrutkovacky.Uhol_ToleranciaMIN.P2_LavaSkrutkaM6:= UDINT_TO_STRING(P2_Srobovanie.STAV.M6_Uhol_ToleranciaMIN);
            Reports.Skrutkovacky.Uhol_ToleranciaMAX.P2_LavaSkrutkaM6:= UDINT_TO_STRING(P2_Srobovanie.STAV.M6_Uhol_ToleranciaMAX);
            Reports.Skrutkovacky.Uhol_NameranaHodnota.P2_LavaSkrutkaM6:= UDINT_TO_STRING(P2_Srobovanie.STAV.M6_DosiahnutyUhol);

            IF NOT SC_P2_StoperSrobovania.Switch1 THEN
                P2_Skrutk_5F_LavaM6_Vysunutie:= STRING_TO_REAL(Reports.Skrutkovacky.VyskaSkrutkovania.P2_LavaSkrutkaM6);
                IF (P2_Skrutk_5F_LavaM6_Vysunutie <= P2_RemPremenne.P2_Srob5F_LavaM6_Vysunutie_HI) AND (P2_Skrutk_5F_LavaM6_Vysunutie >= P2_RemPremenne.P2_Srob5F_LavaM6_Vysunutie_LO)THEN
                    VysunutieSkrutkovacky_OK:= TRUE;
                ELSE
                    VysunutieSkrutkovacky_OK:= FALSE;
                END_IF
                SC_P2_StoperSrobovania.Switch1:= TRUE;
            END_IF

            IF P2_Srobovanie.STAV.Vysledok_Srobovania = 'OK' THEN
                IF VysunutieSkrutkovacky_OK THEN
                    Reports.Skrutkovacky.VyslednyReport.P2_LavaSkrutkaM6:= 'PASS';
                    SC_P2_StoperSrobovania.ResetStep:= TRUE;
                    SC_P2_StoperSrobovania.Step:= 270;
                ELSE
                    Reports.Skrutkovacky.VyslednyReport.P2_LavaSkrutkaM6:= 'FAIL';
                    IF P2_Srobov_M6_Result_OFF THEN
                        SC_P2_StoperSrobovania.ResetStep:= TRUE;
                        SC_P2_StoperSrobovania.Step:= 270;
                    ELSE
                        SC_P2_StoperSrobovania.ResetStep:= TRUE;
                        SC_P2_StoperSrobovania.Step:= 500;
                    END_IF
                END_IF
            ELSIF P2_Srobovanie.STAV.Vysledok_Srobovania = 'NG' THEN
                Reports.Skrutkovacky.VyslednyReport.P2_LavaSkrutkaM6:= 'FAIL';
                IF P2_Srobov_M6_Result_OFF THEN
                    SC_P2_StoperSrobovania.ResetStep:= TRUE;
                    SC_P2_StoperSrobovania.Step:= 270;
                ELSE
                    SC_P2_StoperSrobovania.ResetStep:= TRUE;
                    SC_P2_StoperSrobovania.Step:= 500;
                END_IF
            END_IF

        270:
            SC_P2_StoperSrobovania.StepName:='270 - Automaticky Rezim - modwel 5F zaskrutkuj pravu skrutku M6';
            SC_P2_StoperSrobovania.IdleTime.PT:= T#200ms;
            SC_P2_StoperSrobovania.AlarmTime.PT:= T#5s;

            IF NOT SC_P2_StoperSrobovania.Switch1 THEN
                P2_Srobovanie.STAV.Vysledok_Srobovania:= '';
                P2_StoperSrobovania.OUT.KOM_5F_ZasrobujPravuSkrutkuM6:= TRUE;
                SC_P2_StoperSrobovania.Switch1:= TRUE;
            END_IF

            IF P2_Srobovanie.OUT.KOM_Srobovanie_Ukoncene THEN
                P2_Srobovanie.OUT.KOM_Srobovanie_Ukoncene:= FALSE;
                P2_StoperSrobovania.OUT.KOM_5F_ZasrobujPravuSkrutkuM6:= FALSE;
                IF P2_StoperSrobovania.STAV.Porucha THEN
                    SC_P2_StoperSrobovania.ResetStep:= TRUE;
                    SC_P2_StoperSrobovania.Step:= 500;
                ELSE
                    SC_P2_StoperSrobovania.ResetStep:= TRUE;
                    SC_P2_StoperSrobovania.Step:= 273;
                END_IF
            END_IF

        273:
            SC_P2_StoperSrobovania.StepName:='273 - Automaticky Rezim - modwel 5F kontrola vysledku zaskrutkovania pravej skrutky M6';
            SC_P2_StoperSrobovania.IdleTime.PT:= T#200ms;
            SC_P2_StoperSrobovania.AlarmTime.PT:= T#5s;

            Reports.Skrutkovacky.Moment_ToleranciaMIN.P2_PravaSkrutkaM6:= REAL_TO_STRING(P2_Srobovanie.STAV.M6_Moment_ToleranciaMIN_REAL);
            Reports.Skrutkovacky.Moment_ToleranciaMAX.P2_PravaSkrutkaM6:= REAL_TO_STRING(P2_Srobovanie.STAV.M6_Moment_ToleranciaMAX_REAL);
            Reports.Skrutkovacky.Moment_NameranaHodnota.P2_PravaSkrutkaM6:= REAL_TO_STRING(P2_Srobovanie.STAV.M6_DosiahnutyMoment_REAL);
            Reports.Skrutkovacky.Uhol_ToleranciaMIN.P2_PravaSkrutkaM6:= UDINT_TO_STRING(P2_Srobovanie.STAV.M6_Uhol_ToleranciaMIN);
            Reports.Skrutkovacky.Uhol_ToleranciaMAX.P2_PravaSkrutkaM6:= UDINT_TO_STRING(P2_Srobovanie.STAV.M6_Uhol_ToleranciaMAX);
            Reports.Skrutkovacky.Uhol_NameranaHodnota.P2_PravaSkrutkaM6:= UDINT_TO_STRING(P2_Srobovanie.STAV.M6_DosiahnutyUhol);

            IF NOT SC_P2_StoperSrobovania.Switch1 THEN
                P2_Skrutk_5F_PravaM6_Vysunutie:= STRING_TO_REAL(Reports.Skrutkovacky.VyskaSkrutkovania.P2_PravaSkrutkaM6);
                IF (P2_Skrutk_5F_PravaM6_Vysunutie <= P2_RemPremenne.P2_Srob5F_PravaM6_Vysunutie_HI) AND (P2_Skrutk_5F_PravaM6_Vysunutie >= P2_RemPremenne.P2_Srob5F_PravaM6_Vysunutie_LO)THEN
                    VysunutieSkrutkovacky_OK:= TRUE;
                ELSE
                    VysunutieSkrutkovacky_OK:= FALSE;
                END_IF
                SC_P2_StoperSrobovania.Switch1:= TRUE;
            END_IF

            IF P2_Srobovanie.STAV.Vysledok_Srobovania = 'OK' THEN
                IF VysunutieSkrutkovacky_OK THEN
                    Reports.Skrutkovacky.VyslednyReport.P2_PravaSkrutkaM6:= 'PASS';
                    SC_P2_StoperSrobovania.ResetStep:= TRUE;
                    SC_P2_StoperSrobovania.Step:= 275;
                ELSE
                    Reports.Skrutkovacky.VyslednyReport.P2_PravaSkrutkaM6:= 'FAIL';
                    IF P2_Srobov_M6_Result_OFF THEN
                        SC_P2_StoperSrobovania.ResetStep:= TRUE;
                        SC_P2_StoperSrobovania.Step:= 275;
                    ELSE
                        SC_P2_StoperSrobovania.ResetStep:= TRUE;
                        SC_P2_StoperSrobovania.Step:= 500;
                    END_IF
                END_IF
            ELSIF P2_Srobovanie.STAV.Vysledok_Srobovania = 'NG' THEN
                Reports.Skrutkovacky.VyslednyReport.P2_PravaSkrutkaM6:= 'FAIL';
                IF P2_Srobov_M6_Result_OFF THEN
                    SC_P2_StoperSrobovania.ResetStep:= TRUE;
                    SC_P2_StoperSrobovania.Step:= 275;
                ELSE
                    SC_P2_StoperSrobovania.ResetStep:= TRUE;
                    SC_P2_StoperSrobovania.Step:= 500;
                END_IF
            END_IF

        275:
            SC_P2_StoperSrobovania.StepName:='275 - Automaticky Rezim - modwel 5F presun manipulatora vpred';
            SC_P2_StoperSrobovania.IdleTime.PT:= T#200ms;
            SC_P2_StoperSrobovania.AlarmTime.PT:= T#5s;

            IF NOT SC_P2_StoperSrobovania.Switch1 THEN
                P2_StoperSrobovania.OUT.KOM_PresunManipulator_DOPREDU:= TRUE;
                SC_P2_StoperSrobovania.Switch1:= TRUE;
            END_IF

            IF P2_Srobovanie.OUT.KOM_PresunVPRED_Ukonceny AND NOT P2_Robot.KOM_IN.Stav_RobotPoziciaCakania THEN
                P2_Srobovanie.OUT.KOM_PresunVPRED_Ukonceny:= FALSE;
                P2_StoperSrobovania.OUT.KOM_PresunManipulator_DOPREDU:= FALSE;
                SC_P2_StoperSrobovania.ResetStep:= TRUE;
                SC_P2_StoperSrobovania.Step:= 278;
            END_IF

        278:
            SC_P2_StoperSrobovania.StepName:='278 - Automaticky Rezim - model 5F vystavenie signalu pre robota chod do cakacej pozicie';
            SC_P2_StoperSrobovania.IdleTime.PT:= T#200ms;
            SC_P2_StoperSrobovania.AlarmTime.PT:= T#5s;

            P2_Robot.KOM_OUT.ManipSrobovania_BezpecnaPozicia:= TRUE;

            IF NOT SC_P2_StoperSrobovania.Switch1 THEN
                P2_Robot.KOM_OUT.Presun_CakaciaPozicia:= TRUE;
                SC_P2_StoperSrobovania.Switch1:= TRUE;
            END_IF

            IF P2_Robot.KOM_IN.Stav_RobotPoziciaCakania THEN
                P2_Robot.KOM_OUT.Presun_CakaciaPozicia:= FALSE;
                P2_Robot.STAV.Srobovanie_PrebiehaManipulacia:= FALSE;
                SC_P2_StoperSrobovania.ResetStep:= TRUE;
                SC_P2_StoperSrobovania.Step:= 280;
            END_IF

        280:
            SC_P2_StoperSrobovania.StepName:='280 - Automaticky Rezim - modwel 5F zaskrutkuj lavu skrutku M4';
            SC_P2_StoperSrobovania.IdleTime.PT:= T#200ms;
            SC_P2_StoperSrobovania.AlarmTime.PT:= T#5s;

            IF NOT SC_P2_StoperSrobovania.Switch1 AND P2_Robot.KOM_IN.Stav_RobotBezpPozicia_Srobovanie THEN
                P2_Srobovanie.STAV.Vysledok_Srobovania:= '';
                P2_StoperSrobovania.OUT.KOM_5F_ZasrobujLavuSkrutkuM4:= TRUE;
                SC_P2_StoperSrobovania.Switch1:= TRUE;
            END_IF

            IF P2_Srobovanie.OUT.KOM_Srobovanie_Ukoncene THEN
                P2_Srobovanie.OUT.KOM_Srobovanie_Ukoncene:= FALSE;
                P2_StoperSrobovania.OUT.KOM_5F_ZasrobujLavuSkrutkuM4:= FALSE;
                IF P2_StoperSrobovania.STAV.Porucha THEN
                    SC_P2_StoperSrobovania.ResetStep:= TRUE;
                    SC_P2_StoperSrobovania.Step:= 500;
                ELSE
                    SC_P2_StoperSrobovania.ResetStep:= TRUE;
                    SC_P2_StoperSrobovania.Step:= 283;
                END_IF
            END_IF

        283:
            SC_P2_StoperSrobovania.StepName:='283 - Automaticky Rezim - modwel 5F kontrola vysledku zaskrutkovania lavej skrutky M4';
            SC_P2_StoperSrobovania.IdleTime.PT:= T#200ms;
            SC_P2_StoperSrobovania.AlarmTime.PT:= T#5s;

            Reports.Skrutkovacky.Moment_ToleranciaMIN.P2_LavaSkrutkaM4:= REAL_TO_STRING(P2_Srobovanie.STAV.M4_Moment_ToleranciaMIN_REAL);
            Reports.Skrutkovacky.Moment_ToleranciaMAX.P2_LavaSkrutkaM4:= REAL_TO_STRING(P2_Srobovanie.STAV.M4_Moment_ToleranciaMAX_REAL);
            Reports.Skrutkovacky.Moment_NameranaHodnota.P2_LavaSkrutkaM4:= REAL_TO_STRING(P2_Srobovanie.STAV.M4_DosiahnutyMoment_REAL);
            Reports.Skrutkovacky.Uhol_ToleranciaMIN.P2_LavaSkrutkaM4:= UDINT_TO_STRING(P2_Srobovanie.STAV.M4_Uhol_ToleranciaMIN);
            Reports.Skrutkovacky.Uhol_ToleranciaMAX.P2_LavaSkrutkaM4:= UDINT_TO_STRING(P2_Srobovanie.STAV.M4_Uhol_ToleranciaMAX);
            Reports.Skrutkovacky.Uhol_NameranaHodnota.P2_LavaSkrutkaM4:= UDINT_TO_STRING(P2_Srobovanie.STAV.M4_DosiahnutyUhol);

            IF NOT SC_P2_StoperSrobovania.Switch1 THEN
                P2_Skrutk_5F_LavaM4_Vysunutie:= STRING_TO_REAL(Reports.Skrutkovacky.VyskaSkrutkovania.P2_LavaSkrutkaM4);
                IF (P2_Skrutk_5F_LavaM4_Vysunutie <= P2_RemPremenne.P2_Srob5F_LavaM4_Vysunutie_HI) AND (P2_Skrutk_5F_LavaM4_Vysunutie >= P2_RemPremenne.P2_Srob5F_LavaM4_Vysunutie_LO)THEN
                    VysunutieSkrutkovacky_OK:= TRUE;
                ELSE
                    VysunutieSkrutkovacky_OK:= FALSE;
                END_IF
                SC_P2_StoperSrobovania.Switch1:= TRUE;
            END_IF

            IF P2_Srobovanie.STAV.Vysledok_Srobovania = 'OK' THEN
                IF VysunutieSkrutkovacky_OK THEN
                    Reports.Skrutkovacky.VyslednyReport.P2_LavaSkrutkaM4:= 'PASS';
                    SC_P2_StoperSrobovania.ResetStep:= TRUE;
                    SC_P2_StoperSrobovania.Step:= 285;
                ELSE
                    Reports.Skrutkovacky.VyslednyReport.P2_LavaSkrutkaM4:= 'FAIL';
                    IF P2_Srobov_M4_Result_OFF THEN
                        SC_P2_StoperSrobovania.ResetStep:= TRUE;
                        SC_P2_StoperSrobovania.Step:= 285;
                    ELSE
                        SC_P2_StoperSrobovania.ResetStep:= TRUE;
                        SC_P2_StoperSrobovania.Step:= 500;
                    END_IF
                END_IF
            ELSIF P2_Srobovanie.STAV.Vysledok_Srobovania = 'NG' THEN
                Reports.Skrutkovacky.VyslednyReport.P2_LavaSkrutkaM4:= 'FAIL';
                IF P2_Srobov_M4_Result_OFF THEN
                    SC_P2_StoperSrobovania.ResetStep:= TRUE;
                    SC_P2_StoperSrobovania.Step:= 285;
                ELSE
                    SC_P2_StoperSrobovania.ResetStep:= TRUE;
                    SC_P2_StoperSrobovania.Step:= 500;
                END_IF
            END_IF

        285:
            SC_P2_StoperSrobovania.StepName:='285 - Automaticky Rezim - modwel 5F zaskrutkuj pravu skrutku M4';
            SC_P2_StoperSrobovania.IdleTime.PT:= T#200ms;
            SC_P2_StoperSrobovania.AlarmTime.PT:= T#5s;

            IF NOT SC_P2_StoperSrobovania.Switch1 AND P2_Robot.KOM_IN.Stav_RobotBezpPozicia_Srobovanie THEN
                P2_Srobovanie.STAV.Vysledok_Srobovania:= '';
                P2_StoperSrobovania.OUT.KOM_5F_ZasrobujPravuSkrutkuM4:= TRUE;
                SC_P2_StoperSrobovania.Switch1:= TRUE;
            END_IF

            IF P2_Srobovanie.OUT.KOM_Srobovanie_Ukoncene THEN
                P2_Srobovanie.OUT.KOM_Srobovanie_Ukoncene:= FALSE;
                P2_StoperSrobovania.OUT.KOM_5F_ZasrobujPravuSkrutkuM4:= FALSE;
                IF P2_StoperSrobovania.STAV.Porucha THEN
                    SC_P2_StoperSrobovania.ResetStep:= TRUE;
                    SC_P2_StoperSrobovania.Step:= 500;
                ELSE
                    SC_P2_StoperSrobovania.ResetStep:= TRUE;
                    SC_P2_StoperSrobovania.Step:= 288;
                END_IF
            END_IF

        288:
            SC_P2_StoperSrobovania.StepName:='288 - Automaticky Rezim - modwel 5F kontrola vysledku zaskrutkovania pravej skrutky M4';
            SC_P2_StoperSrobovania.IdleTime.PT:= T#200ms;
            SC_P2_StoperSrobovania.AlarmTime.PT:= T#5s;

            Reports.Skrutkovacky.Moment_ToleranciaMIN.P2_PravaSkrutkaM4:= REAL_TO_STRING(P2_Srobovanie.STAV.M4_Moment_ToleranciaMIN_REAL);
            Reports.Skrutkovacky.Moment_ToleranciaMAX.P2_PravaSkrutkaM4:= REAL_TO_STRING(P2_Srobovanie.STAV.M4_Moment_ToleranciaMAX_REAL);
            Reports.Skrutkovacky.Moment_NameranaHodnota.P2_PravaSkrutkaM4:= REAL_TO_STRING(P2_Srobovanie.STAV.M4_DosiahnutyMoment_REAL);
            Reports.Skrutkovacky.Uhol_ToleranciaMIN.P2_PravaSkrutkaM4:= UDINT_TO_STRING(P2_Srobovanie.STAV.M4_Uhol_ToleranciaMIN);
            Reports.Skrutkovacky.Uhol_ToleranciaMAX.P2_PravaSkrutkaM4:= UDINT_TO_STRING(P2_Srobovanie.STAV.M4_Uhol_ToleranciaMAX);
            Reports.Skrutkovacky.Uhol_NameranaHodnota.P2_PravaSkrutkaM4:= UDINT_TO_STRING(P2_Srobovanie.STAV.M4_DosiahnutyUhol);

            IF NOT SC_P2_StoperSrobovania.Switch1 THEN
                P2_Skrutk_5F_PravaM4_Vysunutie:= STRING_TO_REAL(Reports.Skrutkovacky.VyskaSkrutkovania.P2_PravaSkrutkaM4);
                IF (P2_Skrutk_5F_PravaM4_Vysunutie <= P2_RemPremenne.P2_Srob5F_PravaM4_Vysunutie_HI) AND (P2_Skrutk_5F_PravaM4_Vysunutie >= P2_RemPremenne.P2_Srob5F_PravaM4_Vysunutie_LO)THEN
                    VysunutieSkrutkovacky_OK:= TRUE;
                ELSE
                    VysunutieSkrutkovacky_OK:= FALSE;
                END_IF
                SC_P2_StoperSrobovania.Switch1:= TRUE;
            END_IF

            IF P2_Srobovanie.STAV.Vysledok_Srobovania = 'OK' THEN
                IF VysunutieSkrutkovacky_OK THEN
                    Reports.Skrutkovacky.VyslednyReport.P2_PravaSkrutkaM4:= 'PASS';
                    SC_P2_StoperSrobovania.ResetStep:= TRUE;
                    SC_P2_StoperSrobovania.Step:= 290;
                ELSE
                    Reports.Skrutkovacky.VyslednyReport.P2_PravaSkrutkaM4:= 'FAIL';
                    IF P2_Srobov_M4_Result_OFF THEN
                        SC_P2_StoperSrobovania.ResetStep:= TRUE;
                        SC_P2_StoperSrobovania.Step:= 290;
                    ELSE
                        SC_P2_StoperSrobovania.ResetStep:= TRUE;
                        SC_P2_StoperSrobovania.Step:= 500;
                    END_IF
                END_IF
            ELSIF P2_Srobovanie.STAV.Vysledok_Srobovania = 'NG' THEN
                Reports.Skrutkovacky.VyslednyReport.P2_PravaSkrutkaM4:= 'FAIL';
                IF P2_Srobov_M4_Result_OFF THEN
                    SC_P2_StoperSrobovania.ResetStep:= TRUE;
                    SC_P2_StoperSrobovania.Step:= 290;
                ELSE
                    SC_P2_StoperSrobovania.ResetStep:= TRUE;
                    SC_P2_StoperSrobovania.Step:= 500;
                END_IF
            END_IF
```
